FUNCTION "GestMotore" : Void
{ S7_Optimized_Access := 'TRUE' }
VERSION : 0.2
   VAR_INPUT
      K_Motore : Int;
      K_TipoMotore : Int;
      K_Zona : Int;
   END_VAR

   VAR_TEMP
      PI_Mitsubishi : Struct
         STW : Word;
         ActualSpeed : DInt;
         Current : DInt;
         DCBus : DInt;
         AlarmCode : DInt;
         CurrentPeak : DInt;
         DCBusPeak : DInt;
         Appo7 : DInt;
         Appo8 : DInt;
         Appo9 : DInt;
         Appo10 : DInt;
         Appo11 : DInt;
         Appo12 : DInt;
         Appo13 : DInt;
         Appo14 : DInt;
      END_STRUCT;
      PO_Mitsubishi : Struct
         CTW : Word;
         Speed_SP : DInt;
         Acc : DInt;
         Dec : DInt;
         FStart : DInt;
         Appo5 : DInt;
         Appo6 : DInt;
         Appo7 : DInt;
         Appo8 : DInt;
         Appo9 : DInt;
         Appo10 : DInt;
      END_STRUCT;
      PI_Siemens : Struct
         STW : Word;
         ActualSpeed : Int;
         ActualCurrent : Int;
         ActualTorque : Int;
         WarningCode : Int;
         FaultCode : Int;
      END_STRUCT;
      PO_Siemens : Struct
         CTW : Word;
         Speed : Int;
         Spare01 : Int;
         Spare02 : Int;
         Spare03 : Int;
         Spare04 : Int;
      END_STRUCT;
      PI_Schneider : Struct
         STW : Word;
         ActualSpeed : Int;
         Enrgy : Int;
         Segnalaz_Code : Int;
         Spare_01 : Int;
         Spare_02 : Int;
      END_STRUCT;
      PO_Schneider : Struct
         CTW : Word;
         Speed_SP : Int;
         Acc_SP : Int;
         Dec_SP : Int;
         Spare_01 : Int;
         Spare_02 : Int;
      END_STRUCT;
      PI_Movimot : Struct
         STW1 : Word;
         OutputCurrent : Word;
         STW2 : Word;
      END_STRUCT;
      PO_Movimot : Struct
         CTW : Word;
         Speed : Int;
         AccRich : Int;
      END_STRUCT;
      PI_MoviGear : Struct
         STW : Word;
         Actual_Speed : Int;
         Status_Fault : Int;
         Actual_Torque : Int;
         DI : Word;
      END_STRUCT;
      PO_MoviGear : Struct
         CTW : Word;
         Target_Speed : Int;
         Acceleration : Int;
         Deceleration : Int;
         DO : Word;
      END_STRUCT;
      PI_Danfoss : Struct
         STW : Word;
         ActualSpeed : Int;
         CodAllarme_W1 : Int;
         CodAllarme_W2 : Int;
         CodWarning_W1 : Int;
         CodWarning_W2 : Int;
      END_STRUCT;
      PO_Danfoss : Struct
         CTW : Word;
         Speed : Int;
         AccRich : Int;
         DecRich : Int;
         PCD_Spare01 : Int;
         PCD_Spare02 : Int;
      END_STRUCT;
      PI_INVT : Struct
         PKW01 : Word;
         PKW02 : Word;
         PKW03 : Word;
         PKW04 : Word;
         STW : Word;
         ActualSpeed : Int;
         BusVoltage : Int;
         OutputCurrent : Int;
         FaultCode : Int;
         Sapre1 : Int;
         Sapre2 : Int;
         Sapre3 : Int;
      END_STRUCT;
      PO_INVT : Struct
         PKW01 : Word;
         PKW02 : Word;
         PKW03 : Word;
         PKW04 : Word;
         CTW : Word;
         Speed : Int;
         Spare1 : Int;
         Spare2 : Int;
         Spare3 : Int;
         Spare4 : Int;
         Spare5 : Int;
         Spare6 : Int;
      END_STRUCT;
      PI_Movitrac : Struct
         STW1 : Word;
         ActualSpeed : Int;
         ActualCurrent : Word;
      END_STRUCT;
      PO_MoviTrac : Struct
         CTW : Word;
         Speed : Int;
         Reserved : Int;
      END_STRUCT;
      PI_Nidec : Struct
         STW : Word;   // Status Word
         ActualSpeed : DInt;   // Actual Speed
         ActualCurrent : DInt;   // Actual Current
         ActualDCBus : Int;   // Actual Voltage
         FaultCode : USInt;   // Allarm Code
      END_STRUCT;
      PO_Nidec : Struct
         CTW : Word;   // Control Word
         Speed : DInt;   // Speed Request
         RampAcc : DInt;   // Acceleration Ramp Rerquest
         RampDec : DInt;   // Deceleration Ramp Rerquest
      END_STRUCT;
      TempEnc : Struct
         RcvDaEncoderSick : Struct
            ZSW2_ENC : Word;
            G1_ZSW : Word;
            Position01 : DWord;
            Position02 : DWord;
            Speed : DInt;
         END_STRUCT;
         SendAEncoderSick : Struct
            STW2_ENC : Word;
            G1_STW : Word;
         END_STRUCT;
         RcvDaEncoder_Ottico : Struct
            Posizione : DInt;
            Velocita : Int;
         END_STRUCT;
         RcvDaEncoder_Magnetico : Struct
            Posizione : DInt;
         END_STRUCT;
         arrRecord : Array[0..15] of Byte;
         PosizioneLettaEnc : DInt;
         VelocitaLettaEnc : DInt;
         AppoSetupRich : DInt;
         AppoSetupEncoder : UDInt;
         SpazioUltimoCiclo : DInt;
         AppoScrEncoder : DWord;
      END_STRUCT;
      TempTelem : Struct
         RcvDaEncoder : Struct
            M05_IN_ActPos : DWord;
            Status : Struct
               M10Status_IN_AvvPlaus : Bool;
               M10Status_IN_AvvTemp : Bool;
               M10Status_IN_AvvLiv : Bool;
               M10Status_IN_Avvlaser : Bool;
               M10Status_IN_ErrPlaus : Bool;
               M10Status_IN_ErrTemp : Bool;
               M10Status_IN_ErrLiv : Bool;
               M10Status_IN_ErrLaser : Bool;
               M10Status_IN_Spento : Bool;
               M10Status_IN_RiscaldaOn : Bool;
               M10Status_IN_MF1On : Bool;
               M10Status_IN_MF2On : Bool;
               M10Status_IN_Res1 : Bool;
               M10Status_IN_Res2 : Bool;
               M10Status_IN_Res3 : Bool;
               M10Status_IN_NoDist : Bool;
            END_STRUCT;
         END_STRUCT;
         SendAEncode : Struct
            M05_OUT_Preset : DWord;
            Status : Struct
               M10Status_OUT_Res1 : Bool;
               M10Status_OUT_Res2 : Bool;
               M10Status_OUT_Res3 : Bool;
               M10Status_OUT_Res4 : Bool;
               M10Status_OUT_Res5 : Bool;
               M10Status_OUT_Res6 : Bool;
               M10Status_OUT_Res7 : Bool;
               M10Status_OUT_Res8 : Bool;
               M10Status_OUT_Disabil : Bool;
               M10Status_OUT_Res9 : Bool;
               M10Status_OUT_Res10 : Bool;
               M10Status_OUT_Res11 : Bool;
               M10Status_OUT_Res12 : Bool;
               M10Status_OUT_Res13 : Bool;
               M10Status_OUT_Res14 : Bool;
               M10Status_OUT_Res15 : Bool;
            END_STRUCT;
         END_STRUCT;
         arrRecord : Array[0..15] of Byte;
         AppoSetupRich : DInt;
      END_STRUCT;
      ReqDirPos : Bool;
      ReqDirNeg : Bool;
      FunzPositioning : Bool;
      ReqDecBassa : Bool;
      ReqDecStop : Bool;
      ReqStop : Bool;
      ReqCambioVel : Bool;
      CambioPercLavoro : Bool;
      CambioReqVel : Bool;
      CambioReqAcc : Bool;
      CambioReqDec : Bool;
      REQSetup : Bool;
      REQSetupPannello : Bool;
      DistTrgMagPrec : Bool;
      DistTrgMinPrec : Bool;
      RitMotInPrecisione : Bool;
      UnaDirezioneRichiesta : Bool;
      ReqRicTempoProfilo : Bool;
      BloccaAcc : Bool;
      AbilDirPos : Bool;
      AbilDirNeg : Bool;
      SetUpSuSensore : Bool;
      SetUpFermoMeccanico : Bool;
      RichCmdFreno : Bool;
      SpazioFrenoDir : DInt;
      VeloFrenoDir : DInt;
      AppoMoltPrecisione : DInt;
      DecActRich : DInt;
      RicircoloTotale : DInt;
      MezzoRicircoloTotale : DInt;
      DistCambioVel : DInt;
      SpazioStop : DInt;
      SpazioBassa : DInt;
      SpazioCambioVel : DInt;
      DistTRG_ASS : DInt;
      VeloBassaConv : Real;
      SpazioStop_01 : Real;
      SpazioStop_02 : Real;
      SpazioStop_03 : Real;
      SpazioStop_04 : Real;
      SpazioCambioVel_01 : Real;
      SpazioCambioVel_02 : Real;
      VeloProfilo : Real;
      TempoAcc : Real;
      TempoDec_Iniziale : Real;
      TempoDec_Finale : Real;
      TempoVFix : Real;
      K_MotoreInt : Int;
      K_ZonaInt : Int;
      CounterAllarme : Int;
   END_VAR


BEGIN
	REGION Diagnostica programmatore
	    (*Passiamo tutte le costanti di accesso agli array in modo da verificarle e controllarle*)
	    "Diagnostica"(K_Attuale_ArrayInCuiAccediamo := #K_Motore,
	                  K_NumMax_MassimoValoreDellArrayInCuiAccediamo := "K_NumMotore",
	                  K_Tipo_ArrayInCuiAccediamo := "K_TipoMotore",
	                  K_Attuale_DiChiAccede := #K_Motore,
	                  K_Tipo_DiChiAccede := "K_TipoSezionePastorizzatore",
	                  K_AttualeInterno => #K_MotoreInt);

	    "Diagnostica"(K_Attuale_ArrayInCuiAccediamo := #K_Zona,
	                  K_NumMax_MassimoValoreDellArrayInCuiAccediamo := "K_NumZona",
	                  K_Tipo_ArrayInCuiAccediamo := "K_TipoMotore",
	                  K_Attuale_DiChiAccede := #K_Motore,
	                  K_Tipo_DiChiAccede := "K_TipoMotore",
	                  K_AttualeInterno => #K_ZonaInt);
	END_REGION ;
	REGION From inverter
	    CASE "Motore".M[#K_MotoreInt].HW.TipoCollInverter OF
	        1:
	            REGION PN Mitsubishi
	                (*
	                BIT 00: Drive PI:Ready to Switch ON
	                BIT 01: Drive PI:Ready to Operate
	                BIT 02: Drive PI:Operation Enabled
	                BIT 03: Drive PI:Fault Present
	                BIT 04: Drive PI:Coast Stop
	                BIT 05: Drive PI:Quick Stop
	                BIT 06: Drive PI:Switch ON Inhibited
	                BIT 07: Drive PI:Warning
	                BIT 08:
	                BIT 09: Drive PI: Control ON
	                BIT 10:
	                BIT 11:
	                BIT 12:
	                BIT 13:
	                BIT 14:
	                BIT 15:
	                *)
	                "Motore".M[#K_MotoreInt].Dati.RetVal_Read_Inv := DPRD_DAT(LADDR := "Motore".M[#K_MotoreInt].HW.HWIO_Inverter, RECORD => #PI_Mitsubishi);
	                "Motore".M[#K_MotoreInt].In.NoComunInv := ("Motore".M[#K_MotoreInt].Dati.RetVal_Read_Inv OR "Motore".M[#K_MotoreInt].Dati.RetVal_SCR_Inv) <> 0;
	                IF NOT "Motore".M[#K_MotoreInt].In.NoComunInv THEN
	                    (*Appoggio la Status Word per HMI*)
	                    "Motore".M[#K_MotoreInt].HMI.STW1 := #PI_Mitsubishi.STW;
	                    (*Controllo se l'inverter Ã¨ in Fault e relativo Codice*)
	                    "Motore".M[#K_MotoreInt].In.DriverFault := "Zona".Z[#K_Zona].Out.CentralinaOk AND #PI_Mitsubishi.STW.%X3;
	                    IF "Motore".M[#K_MotoreInt].In.DriverFault THEN
	                        "Motore".M[#K_MotoreInt].HMI.CodiceAllarme := #PI_Mitsubishi.AlarmCode;
	                    END_IF;
	                    (* Calcolo La velocitÃ  letta dall'inverter *)
	                    "Motore".M[#K_MotoreInt].Out.MotorSpeed := TRUNC(ABS(DINT_TO_REAL(#PI_Mitsubishi.ActualSpeed)) * DINT_TO_REAL("Motore".M[#K_MotoreInt].Prm.C.VelMax) / 10000.0);
	                    (* Assegno il segnale di Inverter RUN *)
	                    "Motore".M[#K_MotoreInt].In.MotoreRun := #PI_Mitsubishi.STW.%X2;
	                ELSE
	                    (* In caso di mancanza Comunicazione, Azzero i dati *)
	                    "Motore".M[#K_MotoreInt].Out.MotorSpeed := 0;
	                    "Motore".M[#K_MotoreInt].In.MotoreRun := "Motore".M[#K_MotoreInt].In.DriverFault := "Motore".M[#K_MotoreInt].In.DriverWarning := false;
	                END_IF;
	            END_REGION
	        2:
	            REGION PN Siemens
	                (*
	                Definizione Parola di Stato:
	                Bit 00: Drive PI: Ready TO Switch "ON"
	                Bit 01: Drive PI: Ready TO Operate
	                Bit 02: Drive PI: Operation Enabled. The Drive Follows the Setpoint
	                Bit 03: Drive PI: Fault
	                Bit 04: Drive PI: Coast Stop (OFF2) command is NOT Active
	                Bit 05: Drive PI: Quick Stop (OFF3) command is NOT Active
	                Bit 06: Drive PI: Switching on inhibited
	                Bit 07: Drive PI: Warning
	                Bit 08: Drive PI: Setpoint/Actual Value deviation within tolerance range.
	                Bit 09: Drive PI: Master control requested
	                Bit 10: Drive PI: Maximum frequency reached OR exceeded
	                Bit 11: Drive PI: Motor at Current/Torque limit
	                Bit 12: Drive PI: Motor Holding Brake Open
	                Bit 13: Drive PI: Motor Overload
	                Bit 14: Drive PI: Motor Rotation (1 = CW; 0 = CCW).
	                Bit 15: Drive PI: Inverter Overload
	                *)
	                "Motore".M[#K_MotoreInt].Dati.RetVal_Read_Inv := DPRD_DAT(LADDR := "Motore".M[#K_MotoreInt].HW.HWIO_Inverter, RECORD => #PI_Siemens);
	                "Motore".M[#K_MotoreInt].In.NoComunInv := ("Motore".M[#K_MotoreInt].Dati.RetVal_Read_Inv OR "Motore".M[#K_MotoreInt].Dati.RetVal_SCR_Inv) <> 0;
	                IF NOT "Motore".M[#K_MotoreInt].In.NoComunInv THEN
	                    (*Appoggio la Status Word per HMI*)
	                    "Motore".M[#K_MotoreInt].HMI.STW1 := #PI_Siemens.STW;
	                    (*Controllo se l'inverter Ã¨ in Fault e relativo Codice*)
	                    "Motore".M[#K_MotoreInt].In.DriverFault := "Zona".Z[#K_Zona].Out.CentralinaOk AND (#PI_Siemens.STW.%X3 OR NOT #PI_Siemens.STW.%X9);
	                    IF "Motore".M[#K_MotoreInt].In.DriverFault THEN
	                        "Motore".M[#K_MotoreInt].HMI.CodiceAllarme := #PI_Siemens.FaultCode;
	                    END_IF;
	                    (*Controllo se l'inverter Ã¨ in Warning e relativo Codice*)
	                    "Motore".M[#K_MotoreInt].In.DriverWarning := "Zona".Z[#K_Zona].Out.CentralinaOk AND #PI_Siemens.STW.%X7;
	                    IF "Motore".M[#K_MotoreInt].In.DriverWarning THEN
	                        "Motore".M[#K_MotoreInt].HMI.CodiceWarning := #PI_Siemens.WarningCode;
	                    END_IF;
	                    (* Calcolo La velocitÃ  letta dall'inverter *)
	                    "Motore".M[#K_MotoreInt].Out.MotorSpeed := INT_TO_DINT(#PI_Siemens.ActualSpeed) * "Motore".M[#K_MotoreInt].Prm.C.VelMax / 16384;
	                    (* Assegno il segnale di Inverter RUN *)
	                    "Motore".M[#K_MotoreInt].In.MotoreRun := #PI_Siemens.STW.%X2;
	                ELSE
	                    (* In caso di mancanza Comunicazione, Azzero i dati *)
	                    "Motore".M[#K_MotoreInt].Out.MotorSpeed := 0;
	                    "Motore".M[#K_MotoreInt].In.MotoreRun := "Motore".M[#K_MotoreInt].In.DriverFault := "Motore".M[#K_MotoreInt].In.DriverWarning := false;
	                END_IF;
	            END_REGION
	        3:
	            REGION PN_Schneider
	                (*
	                BIT 00: Drive PI: Mains power supply is switched on, electronics are initialized, pulses are inhibited
	                BIT 01: Drive PI: Refer to control word 1, bit 0
	                BIT 02: Drive PI: Drive follows a reference frequency.
	                BIT 03: Drive PI: An error has been detected.
	                BIT 04: Drive PI: 1= --, 0= Coast stop (OFF 2) command is present
	                BIT 05: Drive PI: 1= --, 0= Quick Stop (OFF 3) command is present.
	                BIT 06: Drive PI: The drive is in Switching on inhibited operating state.
	                BIT 07: Drive PI: Warning information present in the service/maintenance parameter, acknowledgement required.
	                BIT 08: Actual value is within a tolerance band; dynamic speed discrepancies are permissible.
	                BIT 09: The automation system controls the drive.
	                BIT 10: Actual output frequency â‰¥ reference frequency which may be set via the parameter number.
	                BIT 11: Drive PI: Reserved
	                BIT 12: Drive PI: Reserved
	                BIT 13: Drive PI: Reserved
	                BIT 14: Drive PI: Reserved
	                BIT 15: Drive PI: Reserved
	                *)
	                "Motore".M[#K_MotoreInt].Dati.RetVal_Read_Inv := DPRD_DAT(LADDR := "Motore".M[#K_MotoreInt].HW.HWIO_Inverter, RECORD => #PI_Schneider);
	                "Motore".M[#K_MotoreInt].In.NoComunInv := ("Motore".M[#K_MotoreInt].Dati.RetVal_Read_Inv OR "Motore".M[#K_MotoreInt].Dati.RetVal_SCR_Inv) <> 0;
	                IF NOT "Motore".M[#K_MotoreInt].In.NoComunInv THEN
	                    (*Appoggio la Status Word per HMI*)
	                    "Motore".M[#K_MotoreInt].HMI.STW1 := #PI_Schneider.STW;
	                    (*Controllo se l'inverter Ã¨ in Fault e relativo Codice*)
	                    "Motore".M[#K_MotoreInt].In.DriverFault := "Zona".Z[#K_Zona].Out.CentralinaOk AND #PI_Schneider.STW.%X3;
	                    IF "Motore".M[#K_MotoreInt].In.DriverFault THEN
	                        "Motore".M[#K_MotoreInt].HMI.CodiceAllarme := #PI_Schneider.Segnalaz_Code;
	                    END_IF;
	                    // Inverter in warning
	                    "Motore".M[#K_MotoreInt].In.DriverWarning := "Zona".Z[#K_Zona].Out.CentralinaOk AND #PI_Schneider.STW.%X7;
	                    IF "Motore".M[#K_MotoreInt].In.DriverWarning THEN
	                        "Motore".M[#K_MotoreInt].HMI.CodiceWarning := #PI_Schneider.Spare_01;
	                    END_IF;
	                    (* Calcolo La velocitÃ  letta dall'inverter *)
	                    "Motore".M[#K_MotoreInt].Out.MotorSpeed := ABS(INT_TO_DINT(#PI_Schneider.ActualSpeed) * "Motore".M[#K_MotoreInt].Prm.C.VelMax / 3000);
	                    (* Assegno il segnale di Inverter RUN *)
	                    "Motore".M[#K_MotoreInt].In.MotoreRun := #PI_Schneider.STW.%X2;
	                ELSE
	                    (* In caso di mancanza Comunicazione, Azzero i dati *)
	                    "Motore".M[#K_MotoreInt].Out.MotorSpeed := 0;
	                    "Motore".M[#K_MotoreInt].In.MotoreRun := "Motore".M[#K_MotoreInt].In.DriverFault := "Motore".M[#K_MotoreInt].In.DriverWarning := false;
	                END_IF;
	            END_REGION
	        4:
	            REGION PN Movimot
	                (*
	                Status Word 01

	                BIT 08: Alarm Code Bit 00
	                BIT 09: Alarm Code Bit 01
	                BIT 10: Alarm Code Bit 02
	                BIT 11: Alarm Code Bit 03
	                BIT 12: Alarm Code Bit 04
	                BIT 13: Alarm Code Bit 05
	                BIT 14: Alarm Code Bit 06
	                BIT 15: Alarm Code Bit 07
	                BIT 00: 0=Control Not Enabled / 1=Enabled
	                BIT 01: 0=Inverter Not Ready / 1=Ready
	                BIT 02: 0=PO Data Not Enabled / 1=Enabled
	                BIT 03: Reserved
	                BIT 04: Reserved
	                BIT 05: 0=OK / 1=Malfunction/Warning
	                BIT 06: Reserved
	                BIT 07: Reserved

	                Status Word 02

	                BIT 08: 0=Brake Released / 1= Brake Applied
	                BIT 09: 0=Not Ready For Operation / 1=Ready
	                BIT 10: 0=Stop / 1=Motor Run CW
	                BIT 11: 0=Stop / 1=Motor Run CCW
	                BIT 12: 0=Stop / 1=Set Point F2
	                BIT 13: Reserved
	                BIT 14: Reserved
	                BIT 15: Reserved
	                BIT 00: 0=Control Not Enabled / 1=Enabled
	                BIT 01: 0=Inverter Not Ready / 1=Ready
	                BIT 02: 0=PO Data Not Enabled / 1=Enabled
	                BIT 03: Reserved
	                BIT 04: Reserved
	                BIT 05: 0=OK / 1=Malfunction/Warning
	                BIT 06: Reserved
	                BIT 07: Reserved
	                *)
	                "Motore".M[#K_MotoreInt].Dati.RetVal_Read_Inv := DPRD_DAT(LADDR := "Motore".M[#K_MotoreInt].HW.HWIO_Inverter, RECORD => #PI_Movimot);
	                "Motore".M[#K_MotoreInt].In.NoComunInv := ("Motore".M[#K_MotoreInt].Dati.RetVal_Read_Inv OR "Motore".M[#K_MotoreInt].Dati.RetVal_SCR_Inv) <> 0;
	                IF NOT "Motore".M[#K_MotoreInt].In.NoComunInv THEN
	                    (*Appoggio la Status Word per HMI*)
	                    "Motore".M[#K_MotoreInt].HMI.STW1 := #PI_Movimot.STW1;
	                    "Motore".M[#K_MotoreInt].HMI.STW2 := #PI_Movimot.OutputCurrent;
	                    "Motore".M[#K_MotoreInt].HMI.STW3 := #PI_Movimot.STW2;
	                    (* Controllo Stato Sezionatore Aperto *)
	                    "Motore".M[#K_MotoreInt].In.SezAperto := FALSE;
	                    IF #PI_Movimot.STW1.%X5 AND #PI_Movimot.STW1.%X8 AND #PI_Movimot.STW1.%X9 AND #PI_Movimot.STW1.%X10 AND
	                        #PI_Movimot.STW1.%X11 AND NOT #PI_Movimot.STW1.%X12 AND #PI_Movimot.STW1.%X13 AND #PI_Movimot.STW1.%X14 AND
	                        NOT #PI_Movimot.STW1.%X15 AND "Zona".Z[#K_Zona].Out.CentralinaOk THEN
	                        IF "Motore".M[#K_MotoreInt].Dati.ContOffSezAperto < 0 THEN
	                            "Motore".M[#K_MotoreInt].In.SezAperto := TRUE;
	                        ELSE
	                            "Motore".M[#K_MotoreInt].Dati.ContOffSezAperto -= REAL_TO_INT("Zona".Comuni.TempoCicloCpu_r);
	                        END_IF;
	                    ELSE
	                        "Motore".M[#K_MotoreInt].Dati.ContOffSezAperto := 4000;
	                    END_IF;
	                    (*Controllo se l'inverter Ã¨ in Fault e relativo Codice*)
	                    "Motore".M[#K_MotoreInt].In.DriverFault := "Zona".Z[#K_Zona].Out.CentralinaOk AND NOT "Motore".M[#K_MotoreInt].In.SezAperto AND (#PI_Movimot.STW1.%X5 OR NOT #PI_Movimot.STW1.%X1 OR NOT #PI_Movimot.STW1.%X2);
	                    IF "Motore".M[#K_MotoreInt].In.DriverFault THEN
	                        "Motore".M[#K_MotoreInt].HMI.CodiceAllarme := #PI_Movimot.STW1.%B1;
	                    END_IF;
	                    (* Calcolo La velocitÃ  letta dall'inverter *)
	                    "Motore".M[#K_MotoreInt].Out.MotorSpeed := TRUNC("Motore".M[#K_MotoreInt].Out.Vel);
	                    (* Assegno il segnale di Inverter RUN *)
	                    "Motore".M[#K_MotoreInt].In.MotoreRun := #PI_Movimot.STW1.%X0 AND #PI_Movimot.STW2.%X1;
	                ELSE
	                    (* In caso di mancanza Comunicazione, Azzero i dati *)
	                    "Motore".M[#K_MotoreInt].Out.MotorSpeed := 0;
	                    "Motore".M[#K_MotoreInt].In.MotoreRun := "Motore".M[#K_MotoreInt].In.DriverFault := "Motore".M[#K_MotoreInt].In.DriverWarning := false;
	                END_IF;
	            END_REGION
	        5:
	            REGION PN MoviGear
	                (*
	                BIT 00: Ready
	                BIT 01: STO Disattivato
	                BIT 02: Output Stage Pronto
	                BIT 03: Freno Rilasciato
	                BIT 04: Motore in movimento
	                BIT 05: Motore Riferenziato
	                BIT 06: Nuova posizione Relativa Applicata
	                BIT 07: In Posizione
	                BIT 08: Fault
	                BIT 09: Warning
	                BIT 10: Attivato Motore 2
	                BIT 11: VelocitÃ  Attuale = A Target
	                BIT 12: Limiti SW Disattivati
	                BIT 13: Riservato
	                BIT 14: Stand By Attivo
	                BIT 15: HandShake
	                *)
	                "Motore".M[#K_MotoreInt].Dati.RetVal_Read_Inv := DPRD_DAT(LADDR := "Motore".M[#K_MotoreInt].HW.HWIO_Inverter, RECORD => #PI_MoviGear);
	                "Motore".M[#K_MotoreInt].In.NoComunInv := ("Motore".M[#K_MotoreInt].Dati.RetVal_Read_Inv OR "Motore".M[#K_MotoreInt].Dati.RetVal_SCR_Inv) <> 0;
	                IF NOT "Motore".M[#K_MotoreInt].In.NoComunInv THEN
	                    (*Appoggio la Status Word per HMI*)
	                    "Motore".M[#K_MotoreInt].HMI.STW1 := #PI_MoviGear.STW;
	                    (*Controllo se l'inverter Ã¨ in Fault e relativo Codice*)
	                    "Motore".M[#K_MotoreInt].In.DriverFault := "Zona".Z[#K_Zona].Out.CentralinaOk AND (#PI_MoviGear.STW.%X8 OR NOT #PI_MoviGear.STW.%X0);
	                    IF "Motore".M[#K_MotoreInt].In.DriverFault THEN
	                        IF NOT #PI_MoviGear.STW.%X0 THEN
	                            "Motore".M[#K_MotoreInt].HMI.CodiceAllarme := #PI_MoviGear.Status_Fault;
	                        ELSE
	                            "Motore".M[#K_MotoreInt].HMI.CodiceAllarme := 1;
	                        END_IF;
	                    END_IF;
	                    (*Controllo se l'inverter Ã¨ in Warning e relativo Codice*)
	                    "Motore".M[#K_MotoreInt].In.DriverWarning := "Zona".Z[#K_Zona].Out.CentralinaOk AND #PI_MoviGear.STW.%X9;
	                    IF "Motore".M[#K_MotoreInt].In.DriverWarning THEN
	                        "Motore".M[#K_MotoreInt].HMI.CodiceWarning := "Motore".M[#K_MotoreInt].HMI.CodiceWarning;
	                    END_IF;
	                    (* Calcolo La velocitÃ  letta dall'inverter *)
	                    "Motore".M[#K_MotoreInt].Out.MotorSpeed := ABS(INT_TO_DINT(#PI_MoviGear.Actual_Speed)) * "Motore".M[#K_MotoreInt].Prm.C.VelMax / 3000;
	                    (* Assegno il segnale di Inverter RUN *)
	                    "Motore".M[#K_MotoreInt].In.MotoreRun := #PI_MoviGear.STW.%X0 AND #PI_MoviGear.STW.%X2;
	                ELSE
	                    (* In caso di mancanza Comunicazione, Azzero i dati *)
	                    "Motore".M[#K_MotoreInt].Out.MotorSpeed := 0;
	                    "Motore".M[#K_MotoreInt].In.MotoreRun := "Motore".M[#K_MotoreInt].In.DriverFault := "Motore".M[#K_MotoreInt].In.DriverWarning := false;
	                END_IF;
	            END_REGION
	        6:
	            REGION PN Danfoss
	                (*
	                BIT 00: 0=Control NOT Ready       1=Ready
	                BIT 01: 0=Drive NOT Ready       1=Ready
	                BIT 02: 0=Coasting        1=Enable
	                BIT 03: 0=No error        1=Trip
	                BIT 04: OFF/ON 2
	                BIT 05: OFF/ON 3
	                BIT 06: 0=Start possible        1=NOT possible
	                BIT 07: 0=No warning        1=Warning
	                BIT 08: 0= Speed><REF       1= Speed=REF
	                BIT 09: 0=Local oper       1=Bus control
	                BIT 10: 0=Out Freq.Limit     1=Freq.Limit OK
	                BIT 11: 0=No operation      1=In operation
	                BIT 12: 0=Drive OK       1=Stopped, Autostart
	                BIT 13: 0=Voltage OK       1=Voltage exceeded
	                BIT 14: 0=OFF      1=Comparatore 0 ON
	                BIT 15: 0=OFF      1=Comparatore 1 ON
	                *)
	                "Motore".M[#K_MotoreInt].Dati.RetVal_Read_Inv := DPRD_DAT(LADDR := "Motore".M[#K_MotoreInt].HW.HWIO_Inverter, RECORD => #PI_Danfoss);
	                "Motore".M[#K_MotoreInt].In.NoComunInv := ("Motore".M[#K_MotoreInt].Dati.RetVal_Read_Inv OR "Motore".M[#K_MotoreInt].Dati.RetVal_SCR_Inv) <> 0;
	                IF NOT "Motore".M[#K_MotoreInt].In.NoComunInv THEN
	                    (*Appoggio la Status Word per HMI*)
	                    "Motore".M[#K_MotoreInt].HMI.STW1 := #PI_Danfoss.STW;
	                    (*Controllo se l'inverter Ã¨ in Fault e relativo Codice*)
	                    "Motore".M[#K_MotoreInt].In.DriverFault := "Zona".Z[#K_Zona].Out.CentralinaOk AND (#PI_Danfoss.STW.%X3 OR NOT #PI_Danfoss.STW.%X9);
	                    IF "Motore".M[#K_MotoreInt].In.DriverFault THEN
	                        "Motore".M[#K_MotoreInt].HMI.CodiceAllarme := #PI_Danfoss.CodAllarme_W2 OR SHL(IN := #PI_Danfoss.CodAllarme_W1, N := 16);
	                    END_IF;
	                    (*Controllo se l'inverter Ã¨ in Warning e relativo Codice*)
	                    "Motore".M[#K_MotoreInt].In.DriverWarning := "Zona".Z[#K_Zona].Out.CentralinaOk AND #PI_Danfoss.STW.%X7;
	                    IF "Motore".M[#K_MotoreInt].In.DriverWarning THEN
	                        "Motore".M[#K_MotoreInt].HMI.CodiceAllarme := #PI_Danfoss.CodWarning_W2 OR SHL(IN := #PI_Danfoss.CodWarning_W1, N := 16);
	                    END_IF;
	                    (* Calcolo La velocitÃ  letta dall'inverter *)
	                    "Motore".M[#K_MotoreInt].Out.MotorSpeed := ABS(INT_TO_DINT(#PI_Danfoss.ActualSpeed)) * "Motore".M[#K_MotoreInt].Prm.C.VelMax / 16384;
	                    (* Assegno il segnale di Inverter RUN *)
	                    "Motore".M[#K_MotoreInt].In.MotoreRun := #PI_Danfoss.STW.%X2 AND #PI_Danfoss.STW.%X11;
	                ELSE
	                    (* In caso di mancanza Comunicazione, Azzero i dati *)
	                    "Motore".M[#K_MotoreInt].Out.MotorSpeed := 0;
	                    "Motore".M[#K_MotoreInt].In.MotoreRun := "Motore".M[#K_MotoreInt].In.DriverFault := "Motore".M[#K_MotoreInt].In.DriverWarning := false;
	                END_IF;
	            END_REGION
	        7:
	            REGION PN Movitrac
	                (*
	                Status Word 01

	                BIT 08: Alarm Code Bit 00
	                BIT 09: Alarm Code Bit 01
	                BIT 10: Alarm Code Bit 02
	                BIT 11: Alarm Code Bit 03
	                BIT 12: Alarm Code Bit 04
	                BIT 13: Alarm Code Bit 05
	                BIT 14: Alarm Code Bit 06
	                BIT 15: Alarm Code Bit 07
	                BIT 00: 0=Control Not Enabled / 1=Enabled
	                BIT 01: 0=Inverter Not Ready / 1=Ready
	                BIT 02: 0=PO Data Not Enabled / 1=Enabled
	                BIT 03: Reserved
	                BIT 04: Reserved
	                BIT 05: 0=OK / 1=Malfunction/Warning
	                BIT 06: Reserved
	                BIT 07: Reserved
	                *)
	                "Motore".M[#K_MotoreInt].Dati.RetVal_Read_Inv := DPRD_DAT(LADDR := "Motore".M[#K_MotoreInt].HW.HWIO_Inverter, RECORD => #PI_Movitrac);
	                "Motore".M[#K_MotoreInt].In.NoComunInv := ("Motore".M[#K_MotoreInt].Dati.RetVal_Read_Inv OR "Motore".M[#K_MotoreInt].Dati.RetVal_SCR_Inv) <> 0;
	                IF NOT "Motore".M[#K_MotoreInt].In.NoComunInv THEN
	                    (*Appoggio la Status Word per HMI*)
	                    "Motore".M[#K_MotoreInt].HMI.STW1 := #PI_Movitrac.STW1;
	                    (*Controllo se l'inverter Ã¨ in Fault e relativo Codice*)
	                    "Motore".M[#K_MotoreInt].In.DriverFault := "Zona".Z[#K_Zona].Out.CentralinaOk AND (#PI_Movitrac.STW1.%X5 OR NOT #PI_Movitrac.STW1.%X1 OR NOT #PI_Movitrac.STW1.%X2);
	                    IF "Motore".M[#K_MotoreInt].In.DriverFault THEN
	                        "Motore".M[#K_MotoreInt].HMI.CodiceAllarme := #PI_Movitrac.STW1.%B1;
	                    END_IF;
	                    (* Calcolo La velocitÃ  letta dall'inverter *)
	                    "Motore".M[#K_MotoreInt].Out.MotorSpeed := ABS(INT_TO_DINT(#PI_Movitrac.ActualSpeed)) * "Motore".M[#K_MotoreInt].Prm.C.VelMax / 16384;
	                    (* Assegno il segnale di Inverter RUN *)
	                    "Motore".M[#K_MotoreInt].In.MotoreRun := #PI_Movitrac.STW1.%X0;
	                ELSE
	                    (* In caso di mancanza Comunicazione, Azzero i dati *)
	                    "Motore".M[#K_MotoreInt].Out.MotorSpeed := 0;
	                    "Motore".M[#K_MotoreInt].In.MotoreRun := "Motore".M[#K_MotoreInt].In.DriverFault := "Motore".M[#K_MotoreInt].In.DriverWarning := false;
	                END_IF;
	            END_REGION
	        8:
	            REGION PN INVT
	                (*
	                Bit   Descr
	                0â€“7     Running state
	                Value   Desc
	                1       Forward running
	                2       Reverse running
	                3       Stopped
	                4       Faulty
	                5       POFF
	                Bit:8 Bus voltage established: 0=Not ready to Run, 1=Ready to Run
	                Bit 9â€“10: Motor group feedback
	                BIT 11: 0=Asynchronous Motor 1=Syncronous Motor
	                BIT 12:Overload pre-alarm feedback  0=No overload pre-alarm generated 1=Overload pre-alarm generated
	                Bit     Descr
	                13â€“14   Run/Stop mode
	                Value   Desc
	                0       Keypad-based control
	                1       Terminal-based control
	                2       Communication-based control
	                3       Reserved
	                BIT 15Heartbeat feedback : 0=OFF      1=Comparatore 1 ON
	                *)
	                "Motore".M[#K_MotoreInt].Dati.RetVal_Read_Inv := DPRD_DAT(LADDR := "Motore".M[#K_MotoreInt].HW.HWIO_Inverter, RECORD => #PI_INVT);
	                "Motore".M[#K_MotoreInt].In.NoComunInv := ("Motore".M[#K_MotoreInt].Dati.RetVal_Read_Inv OR "Motore".M[#K_MotoreInt].Dati.RetVal_SCR_Inv) <> 0;
	                IF NOT "Motore".M[#K_MotoreInt].In.NoComunInv THEN
	                    (*Appoggio la Status Word per HMI*)
	                    "Motore".M[#K_MotoreInt].HMI.STW1 := #PI_INVT.STW;
	                    (*Controllo se l'inverter Ã¨ in Fault e relativo Codice*)
	                    "Motore".M[#K_MotoreInt].In.DriverFault := #PI_INVT.STW.%B0 = 4 AND "Zona".Z[#K_Zona].Out.CentralinaOk;
	                    IF "Motore".M[#K_MotoreInt].In.DriverFault THEN
	                        "Motore".M[#K_MotoreInt].HMI.CodiceAllarme := #PI_INVT.FaultCode;
	                    END_IF;
	                    (*Controllo se l'inverter Ã¨ in Warning e relativo Codice*)
	                    "Motore".M[#K_MotoreInt].In.DriverWarning := #PI_INVT.STW.%X12;
	                    (* Calcolo La velocitÃ  letta dall'inverter *)
	                    "Motore".M[#K_MotoreInt].Out.MotorSpeed := ABS(INT_TO_DINT(#PI_INVT.ActualSpeed)) * "Motore".M[#K_MotoreInt].Prm.C.VelMax / 10000;
	                    (* Assegno il segnale di Inverter RUN *)
	                    "Motore".M[#K_MotoreInt].In.MotoreRun := #PI_INVT.STW.%X8;
	                ELSE
	                    (* In caso di mancanza Comunicazione, Azzero i dati *)
	                    "Motore".M[#K_MotoreInt].Out.MotorSpeed := 0;
	                    "Motore".M[#K_MotoreInt].In.MotoreRun := "Motore".M[#K_MotoreInt].In.DriverFault := "Motore".M[#K_MotoreInt].In.DriverWarning := false;
	                END_IF;
	            END_REGION
	        9:
	            REGION NIDEC
	                (*
	                BIT 00: Drive Healthy
	                BIT 01: Drive Active
	                BIT 02: Zero Frequency
	                BIT 03: Running At OR Below Minimum Frequency
	                BIT 04: Below Set Frequency
	                BIT 05: At Frequency
	                BIT 06: Above Set Frequency
	                BIT 07: Rated Load Reached
	                BIT 08: Current Limit Active
	                BIT 09: Regenerating
	                BIT 10: Braking IGBT Active
	                BIT 11: Braking Resistor Alarm
	                BIT 12: Reverse Direction Commanded
	                BIT 13: Reverse Direction Running
	                BIT 14: Supply Loss
	                *)
	                IF NOT "Motore".M[#K_MotoreInt].In.NoComunInv THEN
	                    //VariantGet(SRC := #PI_Inv, DST => #PI_Nidec);
	                    "Motore".M[#K_MotoreInt].HMI.STW1 := #PI_Nidec.STW;
	                    (*Controllo se l'inverter Ã¨ in Fault e relativo Codice*)
	                    "Motore".M[#K_MotoreInt].In.DriverFault := NOT #PI_Nidec.STW.%X0 AND "Zona".Z[#K_Zona].Out.CentralinaOk;
	                    IF "Motore".M[#K_MotoreInt].In.DriverFault THEN
	                        "Motore".M[#K_MotoreInt].HMI.CodiceAllarme := #PI_Nidec.FaultCode;
	                    END_IF;
	                    (* Calcolo La velocitÃ  letta dall'inverter *)
	                    "Motore".M[#K_MotoreInt].Out.MotorSpeed := ABS(#PI_Nidec.ActualSpeed) * "Motore".M[#K_MotoreInt].Prm.C.VelMax / 10000;
	                    (* Assegno il segnale di Inverter RUN *)
	                    "Motore".M[#K_MotoreInt].In.MotoreRun := #PI_Nidec.STW.%X1;
	                ELSE
	                    "Motore".M[#K_MotoreInt].Out.MotorSpeed := 0;
	                    "Motore".M[#K_MotoreInt].In.MotoreRun := "Motore".M[#K_MotoreInt].In.DriverFault := "Motore".M[#K_MotoreInt].In.DriverWarning := false;
	                END_IF;
	            END_REGION
	    END_CASE;
	END_REGION
	REGION Encoder manager
	    IF "Zona".Z[#K_Zona].Out.Auto THEN
	        "Motore".M[#K_MotoreInt].HMI.Setup := "Motore".M[#K_MotoreInt].HMI.ManMov := false;
	        "Motore".M[#K_MotoreInt].HMI.ModoInizializza := 0;
	    END_IF;
	    REGION Calcolo Target Position Teorica
	        #RicircoloTotale := "Motore".M[#K_MotoreInt].Prm.Enc.ModuloPosEnc - "Motore".M[#K_MotoreInt].Prm.Enc.ModuloNegEnc;
	        #MezzoRicircoloTotale := #RicircoloTotale / 2;
	        IF "Motore".M[#K_MotoreInt].Out.InMarcia THEN
	            "Motore".M[#K_MotoreInt].Prm.C.TrgPos += "Motore".M[#K_MotoreInt].Out.Vel * "Zona".Comuni.TempoCicloCpu_r / 1000.0;
	            "Motore".M[#K_MotoreInt].Dati.TrgPosDint := TRUNC("Motore".M[#K_MotoreInt].Prm.C.TrgPos);
	            IF "Motore".M[#K_MotoreInt].Prm.Mech.EndLess THEN
	                IF "Motore".M[#K_MotoreInt].Dati.TrgPosDint < "Motore".M[#K_MotoreInt].Prm.Enc.ModuloNegEnc THEN
	                    // Aggiorno l'ultima posizione di target memorizzata
	                    "Motore".M[#K_MotoreInt].Prm.C.TrgPos += DINT_TO_REAL(#RicircoloTotale);
	                    "Motore".M[#K_MotoreInt].Dati.TrgPosDint := "Motore".M[#K_MotoreInt].Dati.OldTrgPosDint := TRUNC("Motore".M[#K_MotoreInt].Prm.C.TrgPos);
	                ELSIF "Motore".M[#K_MotoreInt].Dati.TrgPosDint > "Motore".M[#K_MotoreInt].Prm.Enc.ModuloPosEnc THEN
	                    "Motore".M[#K_MotoreInt].Prm.C.TrgPos -= DINT_TO_REAL(#RicircoloTotale);
	                    "Motore".M[#K_MotoreInt].Dati.TrgPosDint := "Motore".M[#K_MotoreInt].Dati.OldTrgPosDint := TRUNC("Motore".M[#K_MotoreInt].Prm.C.TrgPos);
	                END_IF;
	            END_IF;
	            IF "Motore".M[#K_MotoreInt].Prm.Enc.EncoderLess THEN
	                "Motore".M[#K_MotoreInt].Out.ActPos := "Motore".M[#K_MotoreInt].Dati.TrgPosDint;
	                "Motore".M[#K_MotoreInt].Prm.C.EncPos := "Motore".M[#K_MotoreInt].Prm.C.TrgPos;
	            END_IF;
	        END_IF;
	    END_REGION
	    REGION Condizioni Setup Encoder
	        IF "Motore".M[#K_MotoreInt].In.Setup THEN
	            #REQSetup := TRUE;
	        ELSIF "Motore".M[#K_MotoreInt].HMI.Setup THEN
	            #REQSetupPannello := "Motore".M[#K_MotoreInt].HMI.PulsanteSetupPremuto AND "Zona".Z[#K_Zona].Gen.Reset;
	            IF #REQSetupPannello THEN
	                "Motore".M[#K_MotoreInt].Out.EncoderHomed := FALSE;
	                #SetUpSuSensore := "Motore".M[#K_MotoreInt].Prm.Enc.SetupMode = 2 OR "Motore".M[#K_MotoreInt].Prm.Enc.SetupMode = 10;
	                #SetUpFermoMeccanico := "Motore".M[#K_MotoreInt].Prm.Enc.SetupMode = 4 OR "Motore".M[#K_MotoreInt].Prm.Enc.SetupMode = 12;
	                IF NOT #SetUpSuSensore AND NOT #SetUpFermoMeccanico THEN
	                    #REQSetup := TRUE;
	                    "Motore".M[#K_MotoreInt].Allarmi.SetupEncoderEseg := TRUE;
	                END_IF;
	            END_IF;
	        END_IF;
	    END_REGION
	    REGION Setup Su Sensore
	        IF #SetUpSuSensore OR "Motore".M[#K_MotoreInt].Dati.SetupSensoreTrovato THEN
	            REGION Tempo OFF Marcia Motore
	                IF NOT "Motore".M[#K_MotoreInt].Dati.MotoreFermo THEN
	                    "Motore".M[#K_MotoreInt].Dati.ContTOffMotoreMarcia := 1000;
	                    "Motore".M[#K_MotoreInt].Dati.TOffMotoreMarcia := true;
	                ELSE
	                    IF "Motore".M[#K_MotoreInt].Dati.ContTOffMotoreMarcia > 0 THEN
	                        "Motore".M[#K_MotoreInt].Dati.ContTOffMotoreMarcia -= REAL_TO_INT("Zona".Comuni.TempoCicloCpu_r);
	                    ELSE
	                        "Motore".M[#K_MotoreInt].Dati.TOffMotoreMarcia := false;
	                    END_IF;
	                END_IF;
	            END_REGION ;
	            #REQSetup := "Motore".M[#K_MotoreInt].Out.SetUpSensEseg := "Motore".M[#K_MotoreInt].Dati.SetupSensoreTrovato AND NOT "Motore".M[#K_MotoreInt].Dati.TOffMotoreMarcia;
	            IF #REQSetup THEN
	                "Motore".M[#K_MotoreInt].Allarmi.SetupEncoderEseg := TRUE;
	            END_IF;
	            IF "Motore".M[#K_MotoreInt].Out.SetUpSensEseg THEN
	                IF NOT "Motore".M[#K_MotoreInt].Dati.AppoImpEsecSetUP THEN
	                    "Motore".M[#K_MotoreInt].Dati.Encoder.ValoKSetupSuSens := "Motore".M[#K_MotoreInt].Out.ActPos - "Motore".M[#K_MotoreInt].Dati.PosImpulsoSetup;
	                    "Motore".M[#K_MotoreInt].Dati.AppoImpEsecSetUP := TRUE;
	                END_IF;
	            ELSE
	                "Motore".M[#K_MotoreInt].Dati.AppoImpEsecSetUP := FALSE;
	            END_IF;
	            IF "Motore".M[#K_MotoreInt].Out.SetUpSensEseg AND NOT #SetUpSuSensore THEN
	                IF "Motore".M[#K_MotoreInt].Dati.ContSetUPEncoder > 300 THEN
	                    "Motore".M[#K_MotoreInt].Dati.SetupSensoreTrovato := false;
	                ELSE
	                    "Motore".M[#K_MotoreInt].Dati.ContSetUPEncoder += REAL_TO_INT("Zona".Comuni.TempoCicloCpu_r);
	                END_IF;
	            ELSE
	                "Motore".M[#K_MotoreInt].Dati.ContSetUPEncoder := 0;
	            END_IF;
	            IF NOT "Motore".M[#K_MotoreInt].Dati.SetupSensoreTrovato THEN
	                IF NOT "Motore".M[#K_MotoreInt].In.SensAzz THEN
	                    IF ("Motore".M[#K_MotoreInt].Prm.Enc.SetupMode = 2 AND "Motore".M[#K_MotoreInt].Dati.ActVelNeg) OR
	                        ("Motore".M[#K_MotoreInt].Prm.Enc.SetupMode = 10 AND "Motore".M[#K_MotoreInt].Dati.ActVelPos) THEN
	                        "Motore".M[#K_MotoreInt].Dati.SetupSensoreTrovato := true;
	                        "Motore".M[#K_MotoreInt].Dati.PosImpulsoSetup := "Motore".M[#K_MotoreInt].Out.ActPos;
	                    END_IF;
	                ELSIF ("Motore".M[#K_MotoreInt].Prm.Enc.SetupMode = 2 AND "Motore".M[#K_MotoreInt].Out.ActDirPos) OR
	                    ("Motore".M[#K_MotoreInt].Prm.Enc.SetupMode = 10 AND "Motore".M[#K_MotoreInt].Out.ActDirNeg) THEN
	                    "Motore".M[#K_MotoreInt].Dati.ContTimeOutAzzeramento := 0;
	                END_IF;
	                "Motore".M[#K_MotoreInt].In.CmdPosRich := ("Motore".M[#K_MotoreInt].Prm.Enc.SetupMode = 2 AND NOT "Motore".M[#K_MotoreInt].In.SensAzz) OR ("Motore".M[#K_MotoreInt].Prm.Enc.SetupMode = 10 AND "Motore".M[#K_MotoreInt].In.SensAzz);
	                "Motore".M[#K_MotoreInt].In.CmdNegRich := ("Motore".M[#K_MotoreInt].Prm.Enc.SetupMode = 10 AND NOT "Motore".M[#K_MotoreInt].In.SensAzz) OR ("Motore".M[#K_MotoreInt].Prm.Enc.SetupMode = 2 AND "Motore".M[#K_MotoreInt].In.SensAzz);
	                IF "Motore".M[#K_MotoreInt].In.CmdPosRich THEN
	                    "Motore".M[#K_MotoreInt].In.CmdVelocitaRich := "Motore".M[#K_MotoreInt].Prm.VelSgancioFrenoPos;
	                ELSIF "Motore".M[#K_MotoreInt].In.CmdNegRich THEN
	                    "Motore".M[#K_MotoreInt].In.CmdVelocitaRich := "Motore".M[#K_MotoreInt].Prm.VelSgancioFrenoNeg;
	                END_IF;
	            ELSE
	                "Motore".M[#K_MotoreInt].In.CmdPosRich := "Motore".M[#K_MotoreInt].In.CmdNegRich := "Motore".M[#K_MotoreInt].In.Positioning := false;
	            END_IF;
	        END_IF;
	    END_REGION
	    REGION SetupSuFermoMeccanico
	        IF #SetUpFermoMeccanico OR "Motore".M[#K_MotoreInt].Dati.SetupFermoMeccTrovato THEN
	            REGION Tempo OFF Marcia Motore
	                IF NOT "Motore".M[#K_MotoreInt].Dati.MotoreFermo THEN
	                    "Motore".M[#K_MotoreInt].Dati.ContTOffMotoreMarcia := 1000;
	                    "Motore".M[#K_MotoreInt].Dati.TOffMotoreMarcia := true;
	                ELSE
	                    IF "Motore".M[#K_MotoreInt].Dati.ContTOffMotoreMarcia > 0 THEN
	                        "Motore".M[#K_MotoreInt].Dati.ContTOffMotoreMarcia -= REAL_TO_INT("Zona".Comuni.TempoCicloCpu_r);
	                    ELSE
	                        "Motore".M[#K_MotoreInt].Dati.TOffMotoreMarcia := false;
	                    END_IF;
	                END_IF;
	            END_REGION ;
	            #REQSetup := "Motore".M[#K_MotoreInt].Dati.SetupFermoMeccTrovato AND NOT "Motore".M[#K_MotoreInt].Dati.TOffMotoreMarcia;
	            IF #REQSetup THEN
	                "Motore".M[#K_MotoreInt].Allarmi.SetupEncoderEseg := TRUE;
	            END_IF;
	            IF #REQSetup THEN
	                IF NOT "Motore".M[#K_MotoreInt].Dati.AppoImpEsecSetUP THEN
	                    "Motore".M[#K_MotoreInt].Dati.Encoder.ValoKSetupSuSens := "Motore".M[#K_MotoreInt].Out.ActPos - "Motore".M[#K_MotoreInt].Dati.PosImpulsoSetup;
	                    "Motore".M[#K_MotoreInt].Dati.AppoImpEsecSetUP := TRUE;
	                END_IF;
	            END_IF;
	            IF #REQSetup AND NOT #SetUpFermoMeccanico THEN
	                IF "Motore".M[#K_MotoreInt].Dati.ContSetUPEncoder > 300 THEN
	                    IF NOT #SetUpFermoMeccanico THEN
	                        "Motore".M[#K_MotoreInt].Dati.SetupFermoMeccTrovato := false;
	                    END_IF;
	                ELSE
	                    "Motore".M[#K_MotoreInt].Dati.ContSetUPEncoder += REAL_TO_INT("Zona".Comuni.TempoCicloCpu_r);
	                END_IF;
	            ELSE
	                "Motore".M[#K_MotoreInt].Dati.ContSetUPEncoder := 0;
	            END_IF;
	            IF NOT "Motore".M[#K_MotoreInt].Dati.SetupFermoMeccTrovato THEN
	                "Motore".M[#K_MotoreInt].Dati.AppoImpEsecSetUP := FALSE;
	                IF "Motore".M[#K_MotoreInt].Prm.Enc.SetupMode = 4 THEN
	                    "Motore".M[#K_MotoreInt].In.CmdPosRich := true;
	                    "Motore".M[#K_MotoreInt].In.CmdVelocitaRich := "Motore".M[#K_MotoreInt].Prm.VelSgancioFrenoPos;
	                    IF "Motore".M[#K_MotoreInt].Out.ActDirPos AND "Motore".M[#K_MotoreInt].Out.ActPos <= "Motore".M[#K_MotoreInt].Dati.MaxPosRicercaFermoMeccanico THEN
	                        "Motore".M[#K_MotoreInt].Dati.ContFermoMeccTrovato += REAL_TO_INT("Zona".Comuni.TempoCicloCpu_r);
	                    ELSE
	                        "Motore".M[#K_MotoreInt].Dati.MaxPosRicercaFermoMeccanico := "Motore".M[#K_MotoreInt].Out.ActPos;
	                        "Motore".M[#K_MotoreInt].Dati.ContFermoMeccTrovato := 0;
	                    END_IF;
	                ELSE
	                    "Motore".M[#K_MotoreInt].In.CmdNegRich := true;
	                    "Motore".M[#K_MotoreInt].In.CmdVelocitaRich := "Motore".M[#K_MotoreInt].Prm.VelSgancioFrenoNeg;
	                    IF "Motore".M[#K_MotoreInt].Out.ActDirNeg AND "Motore".M[#K_MotoreInt].Out.ActPos >= "Motore".M[#K_MotoreInt].Dati.MaxPosRicercaFermoMeccanico THEN
	                        "Motore".M[#K_MotoreInt].Dati.ContFermoMeccTrovato += REAL_TO_INT("Zona".Comuni.TempoCicloCpu_r);
	                    ELSE
	                        "Motore".M[#K_MotoreInt].Dati.MaxPosRicercaFermoMeccanico := "Motore".M[#K_MotoreInt].Out.ActPos;
	                        "Motore".M[#K_MotoreInt].Dati.ContFermoMeccTrovato := 0;
	                    END_IF;
	                END_IF;
	                "Motore".M[#K_MotoreInt].Dati.SetupFermoMeccTrovato := "Motore".M[#K_MotoreInt].Dati.ContFermoMeccTrovato > 500;
	                "Motore".M[#K_MotoreInt].Dati.PosImpulsoSetup := "Motore".M[#K_MotoreInt].Dati.MaxPosRicercaFermoMeccanico;
	                "Motore".M[#K_MotoreInt].Dati.ContCheckFollowError := 0;
	            ELSE
	                "Motore".M[#K_MotoreInt].In.CmdPosRich := "Motore".M[#K_MotoreInt].In.CmdNegRich := "Motore".M[#K_MotoreInt].In.Positioning := false;
	            END_IF;
	        END_IF;
	    END_REGION
	    REGION Gestione Encoder
	        (* Gestisco l'Allarme di Setup Eseguito per memorizzare su HMI l'esecuzione del Setuo*)
	        IF "Motore".M[#K_MotoreInt].Allarmi.SetupEncoderEseg THEN
	            "Motore".M[#K_MotoreInt].Dati.ContSegnSetup += REAL_TO_INT("Zona".Comuni.TempoCicloCpu_r);
	            IF "Motore".M[#K_MotoreInt].Dati.ContSegnSetup > 3000 THEN
	                "Motore".M[#K_MotoreInt].Allarmi.SetupEncoderEseg := false;
	                "Motore".M[#K_MotoreInt].Dati.ContSegnSetup := 0;
	            END_IF;
	        END_IF;
	        (* Una volta selezionato su HMI il Setup, se non avviene entro 3 secondi viene deselezionato *)
	        IF "Motore".M[#K_MotoreInt].HMI.Setup AND NOT #REQSetupPannello THEN
	            "Motore".M[#K_MotoreInt].Dati.ContTORichSetup += REAL_TO_INT("Zona".Comuni.TempoCicloCpu_r);
	            IF "Motore".M[#K_MotoreInt].Dati.ContTORichSetup > 3000 THEN
	                "Motore".M[#K_MotoreInt].HMI.Setup := false;
	            END_IF;
	        ELSE
	            "Motore".M[#K_MotoreInt].Dati.ContTORichSetup := 0;
	        END_IF;
	        IF NOT "Motore".M[#K_MotoreInt].Prm.Enc.EncoderLess THEN
	            (* Richiamo la gestione dell'Encoder *)
	            IF "Motore".M[#K_MotoreInt].Prm.Enc.Mounting <> 11 THEN
	                REGION CalcoloPosizioneSetup
	                    IF #REQSetup THEN
	                        CASE "Motore".M[#K_MotoreInt].Prm.Enc.SetupMode OF
	                            0: // Encoder HMI
	                                IF "Motore".M[#K_MotoreInt].Prm.Enc.SetupDoppio THEN
	                                    #TempEnc.AppoSetupRich := "Motore".M[#K_MotoreInt].HMI.ValoreSetupEncoder * 2;
	                                ELSE
	                                    #TempEnc.#AppoSetupRich := "Motore".M[#K_MotoreInt].HMI.ValoreSetupEncoder;
	                                END_IF;
	                                IF NOT "Motore".M[#K_MotoreInt].Prm.Enc.ModoCalcoloK THEN
	                                    "Motore".M[#K_MotoreInt].HMI.ValoreSetupRichiesto := "Motore".M[#K_MotoreInt].Prm.Enc.KSetup + #TempEnc.AppoSetupRich;
	                                ELSE
	                                    "Motore".M[#K_MotoreInt].HMI.ValoreSetupRichiesto := "Motore".M[#K_MotoreInt].Prm.Enc.KSetup - #TempEnc.AppoSetupRich;
	                                END_IF;
	                            1: // Encoder Esterno
	                                "Motore".M[#K_MotoreInt].HMI.ValoreSetupRichiesto := "Motore".M[#K_MotoreInt].In.ValoSetupEnc;
	                            2, 10: // Ricerca Sensore
	                                "Motore".M[#K_MotoreInt].HMI.ValoreSetupRichiesto := "Motore".M[#K_MotoreInt].HMI.ValoreSetupSensore + "Motore".M[#K_MotoreInt].Dati.Encoder.ValoKSetupSuSens;
	                            4, 12: // Ricerca Coppia
	                                "Motore".M[#K_MotoreInt].HMI.ValoreSetupRichiesto := "Motore".M[#K_MotoreInt].HMI.ValoreSetupSensore + "Motore".M[#K_MotoreInt].Dati.Encoder.ValoKSetupSuSens;
	                        END_CASE;
	                    END_IF;
	                END_REGION
	                REGION Lettura Encoder Dal Campo
	                    CASE "Motore".M[#K_MotoreInt].HW.TipoEncoder OF
	                        1:
	                            "Motore".M[#K_MotoreInt].Dati.Encoder.#RetValRdEnc := DPRD_DAT(LADDR := "Motore".M[#K_MotoreInt].HW.HWIO_Encoder, RECORD => #TempEnc.RcvDaEncoderSick);
	                            #TempEnc.#PosizioneLettaEnc := DWORD_TO_DINT(IN := SHR(IN := #TempEnc.RcvDaEncoderSick.Position01, N := 2));
	                            #TempEnc.VelocitaLettaEnc := #TempEnc.RcvDaEncoderSick.Speed;
	                            "Motore".M[#K_MotoreInt].Out.VelEncoder := ABS(TRUNC(DINT_TO_REAL(#TempEnc.VelocitaLettaEnc) * "Motore".M[#K_MotoreInt].Prm.C.SpazioGiroEncoder / "Motore".M[#K_MotoreInt].Prm.Enc.ImpRev * 100.0));
	                            IF (#TempEnc.RcvDaEncoderSick.G1_ZSW.%X15 OR #TempEnc.RcvDaEncoderSick.G1_ZSW.%X12) AND NOT #REQSetup THEN
	                                #TempEnc.SendAEncoderSick.G1_STW := 16#0000;
	                                #TempEnc.SendAEncoderSick.G1_STW.%X15 := #TempEnc.RcvDaEncoderSick.G1_ZSW.%X15;
	                                #TempEnc.SendAEncoderSick.STW2_ENC := 16#400;
	                                "Motore".M[#K_MotoreInt].Dati.Encoder.#RetValScrEnc := DPWR_DAT(LADDR := "Motore".M[#K_MotoreInt].HW.HWIO_Encoder, RECORD := #TempEnc.SendAEncoderSick);
	                            END_IF;
	                        9: // Sick Telemetrica
	                            "Motore".M[#K_MotoreInt].Prm.Enc.Mounting := USint#1;
	                            "Motore".M[#K_MotoreInt].Dati.Encoder.#RetValRdEnc := DPRD_DAT(LADDR := "Motore".M[#K_MotoreInt].HW.HWIO_Encoder, RECORD => #TempTelem.RcvDaEncoder);
	                            "Motore".M[#K_MotoreInt].Dati.Encoder.#RetValRdEnc := DPRD_DAT(LADDR := "Motore".M[#K_MotoreInt].HW.HWIO_PrmEncoder, RECORD => #TempTelem.RcvDaEncoder.Status);
	                            // Valore arriva in decimi di mm (*100 = converto in millesimi di millimetro)
	                            #TempEnc.#PosizioneLettaEnc := DWORD_TO_DINT(#TempTelem.RcvDaEncoder.M05_IN_ActPos * 100);
	                        10:
	                            "Motore".M[#K_MotoreInt].Dati.Encoder.#RetValRdEnc := DPRD_DAT(LADDR := "Motore".M[#K_MotoreInt].HW.HWIO_Encoder, RECORD => #TempEnc.#RcvDaEncoder_Ottico);
	                            #TempEnc.#PosizioneLettaEnc := #TempEnc.#RcvDaEncoder_Ottico.Posizione;
	                        11:
	                            "Motore".M[#K_MotoreInt].Dati.Encoder.#RetValRdEnc := DPRD_DAT(LADDR := "Motore".M[#K_MotoreInt].HW.HWIO_Encoder, RECORD => #TempEnc.#RcvDaEncoder_Magnetico);
	                            #TempEnc.#PosizioneLettaEnc := #TempEnc.#RcvDaEncoder_Magnetico.Posizione;
	                    END_CASE;
	                    "Motore".M[#K_MotoreInt].In.NoComunEnc := "Motore".M[#K_MotoreInt].Dati.Encoder.#RetValRdEnc <> 0 OR #TempEnc.#PosizioneLettaEnc = 0;
	                END_REGION
	                IF NOT "Motore".M[#K_MotoreInt].Prm.Mech.EndLess THEN
	                    REGION Gestione Encoder
	                        REGION CalcoloPosizione
	                            IF NOT "Motore".M[#K_MotoreInt].In.NoComunEnc THEN
	                                IF NOT "Motore".M[#K_MotoreInt].Prm.Enc.Direction THEN
	                                    IF "Motore".M[#K_MotoreInt].HW.TipoEncoder = 9 THEN
	                                        // Se Telemetrica (=9) Cambio Calcolo
	                                        IF #TempEnc.PosizioneLettaEnc <> 0 THEN
	                                            "Motore".M[#K_MotoreInt].Prm.C.EncPos := DINT_TO_REAL(#TempEnc.#PosizioneLettaEnc);
	                                        ELSE
	                                            "Motore".M[#K_MotoreInt].Allarmi.EncMismatch := true;
	                                        END_IF;
	                                    ELSE
	                                        "Motore".M[#K_MotoreInt].Prm.C.EncPos := DINT_TO_REAL(#TempEnc.PosizioneLettaEnc - "Motore".M[#K_MotoreInt].Dati.Encoder.MezzoRicircoloEncoder) / "Motore".M[#K_MotoreInt].Prm.Enc.ImpRev * "Motore".M[#K_MotoreInt].Prm.C.SpazioGiroEncoder;
	                                    END_IF;
	                                ELSE
	                                    IF "Motore".M[#K_MotoreInt].HW.TipoEncoder = 9 THEN
	                                        // Se Telemetrica (=9) Cambio Calcolo
	                                        IF #TempEnc.PosizioneLettaEnc <> 0 THEN
	                                            "Motore".M[#K_MotoreInt].Prm.C.EncPos := DINT_TO_REAL("Motore".M[#K_MotoreInt].Prm.Enc.KSetup - #TempEnc.#PosizioneLettaEnc);
	                                        ELSE
	                                            "Motore".M[#K_MotoreInt].Allarmi.EncMismatch := true;
	                                        END_IF;
	                                    ELSE
	                                        "Motore".M[#K_MotoreInt].Prm.C.EncPos := DINT_TO_REAL(- #TempEnc.PosizioneLettaEnc + "Motore".M[#K_MotoreInt].Dati.Encoder.MezzoRicircoloEncoder) / "Motore".M[#K_MotoreInt].Prm.Enc.ImpRev * "Motore".M[#K_MotoreInt].Prm.C.SpazioGiroEncoder;
	                                    END_IF;
	                                END_IF;
	                            END_IF;
	                        END_REGION
	                        REGION Gestione Setup Encoder
	                            IF #REQSetup THEN
	                                IF NOT "Motore".M[#K_MotoreInt].Dati.Encoder.RichSetupEnc THEN
	                                    "Motore".M[#K_MotoreInt].Out.EncoderHomed := false;
	                                END_IF;
	                                IF NOT "Motore".M[#K_MotoreInt].Prm.Enc.Direction THEN
	                                    #TempEnc.#AppoSetupEncoder := DINT_TO_UDINT(TRUNC(DINT_TO_REAL("Motore".M[#K_MotoreInt].HMI.ValoreSetupRichiesto) / "Motore".M[#K_MotoreInt].Prm.C.SpazioGiroEncoder * "Motore".M[#K_MotoreInt].Prm.Enc.ImpRev) + "Motore".M[#K_MotoreInt].Dati.Encoder.MezzoRicircoloEncoder);
	                                ELSE
	                                    #TempEnc.#AppoSetupEncoder := DINT_TO_UDINT(TRUNC(DINT_TO_REAL(- "Motore".M[#K_MotoreInt].HMI.ValoreSetupRichiesto) / "Motore".M[#K_MotoreInt].Prm.C.SpazioGiroEncoder * "Motore".M[#K_MotoreInt].Prm.Enc.ImpRev) + "Motore".M[#K_MotoreInt].Dati.Encoder.MezzoRicircoloEncoder);
	                                END_IF;
	                                IF "Motore".M[#K_MotoreInt].HW.TipoEncoder = 9 THEN
	                                    IF NOT "Motore".M[#K_MotoreInt].Prm.Enc.ModoCalcoloK THEN
	                                        #TempEnc.#AppoSetupEncoder := DINT_TO_UDINT("Motore".M[#K_MotoreInt].HMI.ValoreSetupRichiesto);
	                                    ELSE
	                                        #TempEnc.#AppoSetupEncoder := DINT_TO_UDINT("Motore".M[#K_MotoreInt].HMI.ValoreSetupEncoder);
	                                    END_IF;
	                                END_IF;
	                                IF #TempEnc.PosizioneLettaEnc <> #TempEnc.#AppoSetupEncoder OR #TempEnc.RcvDaEncoderSick.G1_ZSW.%X12 THEN
	                                    CASE "Motore".M[#K_MotoreInt].HW.TipoEncoder OF
	                                        1:
	                                            #TempEnc.#arrRecord[0] := 1;
	                                            #TempEnc.#arrRecord[1] := 2; (*Request ID = Change parameter*)
	                                            #TempEnc.#arrRecord[2] := 0; (*DO-ID*)
	                                            #TempEnc.#arrRecord[3] := 1; (*No. of parameters*)
	                                            #TempEnc.#arrRecord[4] := 16#10; (*Attribute = Value*)
	                                            #TempEnc.#arrRecord[5] := 0; (*No. of elements*)
	                                            #TempEnc.#arrRecord[6] := 16#fd; (*PNU high byte*)
	                                            #TempEnc.#arrRecord[7] := 16#e8; (*PNU low byte*)
	                                            #TempEnc.#arrRecord[8] := 0; (*Subindex high byte*)
	                                            #TempEnc.#arrRecord[9] := 0; (*Subindex low byte*)
	                                            #TempEnc.#arrRecord[10] := 16#43;
	                                            #TempEnc.#arrRecord[11] := 1;
	                                            #TempEnc.#arrRecord[12] := #TempEnc.#AppoSetupEncoder.%B3;
	                                            #TempEnc.#arrRecord[13] := #TempEnc.#AppoSetupEncoder.%B2;
	                                            #TempEnc.#arrRecord[14] := #TempEnc.#AppoSetupEncoder.%B1;
	                                            #TempEnc.#arrRecord[15] := #TempEnc.#AppoSetupEncoder.%B0;

	                              "WRREC"(REQ := "Motore".M[#K_MotoreInt].Dati.Encoder.RichSetupEnc AND NOT "Motore".M[#K_MotoreInt].Dati.SetupPN.Output.BUSY AND NOT "Motore".M[#K_MotoreInt].Dati.SetupPN.Output.DONE AND NOT "Motore".M[#K_MotoreInt].Dati.Encoder.PrmEncSend,
	                                      ID := "Motore".M[#K_MotoreInt].HW.HWIO_PrmEncoder,
	                                      INDEX := 16#B02E,
	                                      LEN := 16,
	                                      DONE => "Motore".M[#K_MotoreInt].Dati.SetupPN.Output.DONE,
	                                      BUSY => "Motore".M[#K_MotoreInt].Dati.SetupPN.Output.BUSY,
	                                      ERROR => "Motore".M[#K_MotoreInt].Dati.SetupPN.Output.ERROR,
	                                      STATUS => "Motore".M[#K_MotoreInt].Dati.SetupPN.Output.STATUS,
	                                      RECORD := #TempEnc.#arrRecord);

	                              IF "Motore".M[#K_MotoreInt].Dati.Encoder.RichSetupEnc THEN
	                                  IF "Motore".M[#K_MotoreInt].Dati.SetupPN.Output.DONE THEN
	                                                    "Motore".M[#K_MotoreInt].Dati.Encoder.PrmEncSend := true;
	                                                END_IF;
	                                            ELSE
	                                                "Motore".M[#K_MotoreInt].Dati.Encoder.PrmEncSend := false;
	                                            END_IF;
	                                            IF "Motore".M[#K_MotoreInt].Dati.Encoder.PrmEncSend AND NOT #TempEnc.RcvDaEncoderSick.G1_ZSW.%X12 THEN
	                                                #TempEnc.SendAEncoderSick.G1_STW := 16#1000;
	                                            ELSE
	                                                #TempEnc.SendAEncoderSick.G1_STW := 0;
	                                            END_IF;
	                                            #TempEnc.SendAEncoderSick.STW2_ENC := 16#400;
	                                            "Motore".M[#K_MotoreInt].Dati.Encoder.#RetValScrEnc := DPWR_DAT(LADDR := "Motore".M[#K_MotoreInt].HW.HWIO_Encoder, RECORD := #TempEnc.SendAEncoderSick);
	                                        9: // Setup Telemetrica
	                                            // Divido Valore per 100 per scrivere Valore in Decimi di mm
	                                            #TempTelem.SendAEncode.M05_OUT_Preset := UDINT_TO_DWORD(IN := #TempEnc.#AppoSetupEncoder / 100);
	                                            // Alzo bit richiesta Setup
	                                            #TempTelem.SendAEncode.M05_OUT_Preset.%X31 := TRUE;
	                                            "Motore".M[#K_MotoreInt].Dati.Encoder.#RetValScrEnc := DPWR_DAT(LADDR := "Motore".M[#K_MotoreInt].HW.HWIO_Encoder, RECORD := #TempTelem.SendAEncode);
	                                            "Motore".M[#K_MotoreInt].Dati.Encoder.#RichSetupEnc := true;
	                                        10:
	                                            #TempEnc.#AppoScrEncoder := (#TempEnc.#AppoSetupEncoder) OR dw#16#C0000000;

	                              "WRREC"(REQ := "Motore".M[#K_MotoreInt].Dati.Encoder.RichSetupEnc AND NOT "Motore".M[#K_MotoreInt].Dati.SetupPN.Output.BUSY AND NOT "Motore".M[#K_MotoreInt].Dati.SetupPN.Output.DONE,
	                                      ID := "Motore".M[#K_MotoreInt].HW.HWIO_PrmEncoder,
	                                      INDEX := 2,
	                                      LEN := 4,
	                                      DONE => "Motore".M[#K_MotoreInt].Dati.SetupPN.Output.DONE,
	                                      BUSY => "Motore".M[#K_MotoreInt].Dati.SetupPN.Output.BUSY,
	                                      ERROR => "Motore".M[#K_MotoreInt].Dati.SetupPN.Output.ERROR,
	                                      STATUS => "Motore".M[#K_MotoreInt].Dati.SetupPN.Output.STATUS,
	                                      RECORD := #TempEnc.AppoScrEncoder);

	                                        11:
	                                            #TempEnc.#AppoScrEncoder := #TempEnc.#AppoSetupEncoder;
	                                            "WRREC"(REQ := "Motore".M[#K_MotoreInt].Dati.Encoder.RichSetupEnc AND NOT "Motore".M[#K_MotoreInt].Dati.SetupPN.Output.BUSY AND NOT "Motore".M[#K_MotoreInt].Dati.SetupPN.Output.DONE,
	                                                    ID := "Motore".M[#K_MotoreInt].HW.HWIO_PrmEncoder,
	                                                    INDEX := 2,
	                                                    LEN := 4,
	                                                    DONE => "Motore".M[#K_MotoreInt].Dati.SetupPN.Output.DONE,
	                                                    BUSY => "Motore".M[#K_MotoreInt].Dati.SetupPN.Output.BUSY,
	                                                    ERROR => "Motore".M[#K_MotoreInt].Dati.SetupPN.Output.ERROR,
	                                                    STATUS => "Motore".M[#K_MotoreInt].Dati.SetupPN.Output.STATUS,
	                                                    RECORD := #TempEnc.AppoScrEncoder);

	                                    END_CASE;
	                                    "Motore".M[#K_MotoreInt].Dati.Encoder.#RichSetupEnc := true;
	                                ELSE
	                                    "Motore".M[#K_MotoreInt].Out.EncoderHomed := true;
	                                END_IF;
	                            ELSE
	                                IF "Motore".M[#K_MotoreInt].Dati.Encoder.RichSetupEnc THEN
	                                    CASE "Motore".M[#K_MotoreInt].HW.TipoEncoder OF
	                                        9:
	                                            #TempTelem.SendAEncode.M05_OUT_Preset := 0;
	                                            "Motore".M[#K_MotoreInt].Dati.Encoder.#RetValScrEnc := DPWR_DAT(LADDR := "Motore".M[#K_MotoreInt].HW.HWIO_Encoder, RECORD := #TempTelem.SendAEncode);
	                                    END_CASE;
	                                    "Motore".M[#K_MotoreInt].Dati.Encoder.RichSetupEnc := false;
	                                END_IF;
	                            END_IF;
	                        END_REGION
	                    END_REGION
	                ELSE
	                    REGION Gestione Encoder EndLess
	                        REGION Gestione Setup Encoder
	                            IF #REQSetup THEN
	                                "Motore".M[#K_MotoreInt].Out.EncoderHomed := true;
	                                "Motore".M[#K_MotoreInt].Prm.C.EncPos := DINT_TO_REAL("Motore".M[#K_MotoreInt].HMI.ValoreSetupRichiesto);
	                                "Motore".M[#K_MotoreInt].In.Setup := false;
	                            END_IF;
	                        END_REGION
	                        REGION REGION CalcoloPosizione
	                            IF NOT "Motore".M[#K_MotoreInt].In.NoComunEnc THEN
	                                #TempEnc.SpazioUltimoCiclo := #TempEnc.PosizioneLettaEnc - "Motore".M[#K_MotoreInt].Dati.Encoder.o_OldPosEncoder;
	                                IF #TempEnc.SpazioUltimoCiclo <> 0 THEN
	                                    IF ABS(#TempEnc.SpazioUltimoCiclo) > "Motore".M[#K_MotoreInt].Dati.Encoder.#MezzoRicircoloEncoder THEN
	                                        IF #TempEnc.PosizioneLettaEnc < "Motore".M[#K_MotoreInt].Dati.Encoder.o_OldPosEncoder THEN
	                                            #TempEnc.SpazioUltimoCiclo := "Motore".M[#K_MotoreInt].Dati.Encoder.#RicircoloEncoder - "Motore".M[#K_MotoreInt].Dati.Encoder.o_OldPosEncoder + #TempEnc.PosizioneLettaEnc;
	                                        ELSE
	                                            #TempEnc.SpazioUltimoCiclo := #TempEnc.PosizioneLettaEnc - "Motore".M[#K_MotoreInt].Dati.Encoder.#RicircoloEncoder - "Motore".M[#K_MotoreInt].Dati.Encoder.o_OldPosEncoder;
	                                        END_IF;
	                                    END_IF;
	                                    "Motore".M[#K_MotoreInt].Dati.Encoder.o_OldPosEncoder := #TempEnc.PosizioneLettaEnc;
	                                    IF NOT "Motore".M[#K_MotoreInt].Prm.Enc.Direction THEN
	                                        "Motore".M[#K_MotoreInt].Prm.C.EncPos += DINT_TO_REAL(#TempEnc.SpazioUltimoCiclo) * "Motore".M[#K_MotoreInt].Prm.C.SpazioGiroEncoder / "Motore".M[#K_MotoreInt].Prm.Enc.ImpRev;
	                                    ELSE
	                                        "Motore".M[#K_MotoreInt].Prm.C.EncPos -= DINT_TO_REAL(#TempEnc.SpazioUltimoCiclo) * "Motore".M[#K_MotoreInt].Prm.C.SpazioGiroEncoder / "Motore".M[#K_MotoreInt].Prm.Enc.ImpRev;
	                                    END_IF;
	                                    IF "Motore".M[#K_MotoreInt].Prm.C.EncPos > DINT_TO_REAL("Motore".M[#K_MotoreInt].Prm.Enc.ModuloPosEnc) THEN
	                                        "Motore".M[#K_MotoreInt].Prm.C.EncPos -= DINT_TO_REAL("Motore".M[#K_MotoreInt].Prm.Enc.ModuloPosEnc - "Motore".M[#K_MotoreInt].Prm.Enc.ModuloNegEnc);
	                                    ELSIF "Motore".M[#K_MotoreInt].Prm.C.EncPos < DINT_TO_REAL("Motore".M[#K_MotoreInt].Prm.Enc.ModuloNegEnc) THEN
	                                        "Motore".M[#K_MotoreInt].Prm.C.EncPos += DINT_TO_REAL("Motore".M[#K_MotoreInt].Prm.Enc.ModuloPosEnc - "Motore".M[#K_MotoreInt].Prm.Enc.ModuloNegEnc);
	                                    END_IF;
	                                END_IF;
	                            END_IF;
	                        END_REGION
	                    END_REGION
	                END_IF;
	            END_IF;
	            (* Assegnazione dati Posizione Encoder *)
	            "Motore".M[#K_MotoreInt].Out.ActPos := TRUNC("Motore".M[#K_MotoreInt].Prm.C.EncPos);
	            IF #REQSetup THEN
	                "Motore".M[#K_MotoreInt].Dati.PosizioneAlloStop := "Motore".M[#K_MotoreInt].Dati.PosizioneCheckDirezione := "Motore".M[#K_MotoreInt].Dati.TrgPosDint := "Motore".M[#K_MotoreInt].Dati.OldTrgPosDint := "Motore".M[#K_MotoreInt].Dati.OldEncoder := "Motore".M[#K_MotoreInt].Out.ActPos;
	                "Motore".M[#K_MotoreInt].Prm.C.TrgPos := "Motore".M[#K_MotoreInt].Prm.C.EncPos;
	            END_IF;
	        ELSIF #REQSetup THEN
	            (* Gestione Posizione Encoder Simulata *)
	            "Motore".M[#K_MotoreInt].Dati.PosizioneAlloStop := "Motore".M[#K_MotoreInt].Dati.PosizioneCheckDirezione := "Motore".M[#K_MotoreInt].Dati.TrgPosDint := "Motore".M[#K_MotoreInt].Dati.OldTrgPosDint := "Motore".M[#K_MotoreInt].Dati.OldEncoder := "Motore".M[#K_MotoreInt].Out.ActPos := "Motore".M[#K_MotoreInt].HMI.ValoreSetupEncoder;
	            "Motore".M[#K_MotoreInt].Prm.C.TrgPos := "Motore".M[#K_MotoreInt].Prm.C.EncPos := DINT_TO_REAL("Motore".M[#K_MotoreInt].HMI.ValoreSetupEncoder);
	            "Motore".M[#K_MotoreInt].In.Setup := false;
	        END_IF;
	    END_REGION
	    REGION Spazio Ciclo PLC
	        IF "Motore".M[#K_MotoreInt].Out.ActPos <> "Motore".M[#K_MotoreInt].Dati.OldEncoder THEN
	            "Motore".M[#K_MotoreInt].Out.SpazioCicloEnc := "Motore".M[#K_MotoreInt].Out.ActPos - "Motore".M[#K_MotoreInt].Dati.OldEncoder;
	            IF "Motore".M[#K_MotoreInt].Prm.Mech.EndLess THEN
	                IF ABS("Motore".M[#K_MotoreInt].Out.SpazioCicloEnc) > #MezzoRicircoloTotale THEN
	                    IF "Motore".M[#K_MotoreInt].Dati.OldEncoder > "Motore".M[#K_MotoreInt].Out.ActPos THEN
	                        "Motore".M[#K_MotoreInt].Out.SpazioCicloEnc := "Motore".M[#K_MotoreInt].Prm.Enc.ModuloPosEnc - "Motore".M[#K_MotoreInt].Dati.OldEncoder - "Motore".M[#K_MotoreInt].Prm.Enc.ModuloNegEnc + "Motore".M[#K_MotoreInt].Out.ActPos;
	                    ELSE
	                        "Motore".M[#K_MotoreInt].Out.SpazioCicloEnc := "Motore".M[#K_MotoreInt].Out.ActPos - "Motore".M[#K_MotoreInt].Prm.Enc.ModuloPosEnc + "Motore".M[#K_MotoreInt].Prm.Enc.ModuloNegEnc - "Motore".M[#K_MotoreInt].Dati.OldEncoder;
	                    END_IF;
	                END_IF;
	            END_IF;
	            "Motore".M[#K_MotoreInt].Dati.OldEncoder := "Motore".M[#K_MotoreInt].Out.ActPos;
	        ELSE
	            "Motore".M[#K_MotoreInt].Out.SpazioCicloEnc := 0;
	        END_IF;
	    END_REGION
	END_REGION ;
	REGION Limits
	    "Motore".M[#K_MotoreInt].Allarmi.Parametri := false;
	    REGION Abilita Cambio Direzione
	        IF "Motore".M[#K_MotoreInt].Prm.TCambioDir = 0 OR "Motore".M[#K_MotoreInt].Prm.CambioDirNoFreno THEN
	            #AbilDirPos := #AbilDirNeg := true;
	            "Motore".M[#K_MotoreInt].Dati.ContCambioDirPos := "Motore".M[#K_MotoreInt].Dati.ContCambioDirNeg := -1;
	        ELSE
	            IF "Motore".M[#K_MotoreInt].Out.ActDirNeg THEN
	                "Motore".M[#K_MotoreInt].Dati.ContCambioDirPos := "Motore".M[#K_MotoreInt].Prm.TCambioDir;
	            ELSIF "Motore".M[#K_MotoreInt].Out.ActDirPos THEN
	                "Motore".M[#K_MotoreInt].Dati.ContCambioDirNeg := "Motore".M[#K_MotoreInt].Prm.TCambioDir;
	            END_IF;
	            IF "Motore".M[#K_MotoreInt].Dati.ContCambioDirPos < 0 THEN
	                #AbilDirPos := true;
	            ELSE
	                "Motore".M[#K_MotoreInt].Dati.ContCambioDirPos -= REAL_TO_INT("Zona".Comuni.TempoCicloCpu_r);
	                #AbilDirPos := false;
	            END_IF;
	            IF "Motore".M[#K_MotoreInt].Dati.ContCambioDirNeg < 0 THEN
	                #AbilDirNeg := true;
	            ELSE
	                "Motore".M[#K_MotoreInt].Dati.ContCambioDirNeg -= REAL_TO_INT("Zona".Comuni.TempoCicloCpu_r);
	                #AbilDirNeg := false;
	            END_IF;
	        END_IF;
	    END_REGION
	    IF NOT "Motore".M[#K_MotoreInt].Prm.EscludiFunzPos THEN
	        REGION Abilita movimento motore / Posizionamento
	            "Motore".M[#K_MotoreInt].Out.Pronto := FALSE;
	            IF "Zona".Z[#K_Zona].Out.CentralinaOk THEN
	                IF NOT "Motore".M[#K_MotoreInt].In.SezAperto AND NOT "Motore".M[#K_MotoreInt].In.DriverFault AND NOT "Motore".M[#K_MotoreInt].In.NoComunInv THEN
	                    IF NOT "Motore".M[#K_MotoreInt].In.TerVentolaOff AND NOT "Motore".M[#K_MotoreInt].In.CinghiaRotta AND NOT "Motore".M[#K_MotoreInt].In.SpinaSicNoInPos AND ("Motore".M[#K_MotoreInt].In.AnticadutaON OR NOT "Motore".M[#K_MotoreInt].Prm.AnticadutaPresente) THEN
	                        "Motore".M[#K_MotoreInt].Out.Pronto := NOT "Motore".M[#K_MotoreInt].Dati.MotorStop;
	                    ELSIF "Zona".Z[#K_ZonaInt].Out.Man AND "Zona".Z[#K_ZonaInt].Gen.Reset AND ("Motore".M[#K_MotoreInt].In.CmdPosRich OR "Motore".M[#K_MotoreInt].In.CmdNegRich) THEN
	                        "Motore".M[#K_MotoreInt].Out.Pronto := TRUE;
	                    END_IF;
	                END_IF;
	            END_IF;
	            IF "Motore".M[#K_MotoreInt].In.Positioning THEN
	                #FunzPositioning := NOT "Motore".M[#K_MotoreInt].In.CmdPosRich AND NOT "Motore".M[#K_MotoreInt].In.CmdNegRich AND NOT #REQSetupPannello AND "Motore".M[#K_MotoreInt].Out.Pronto AND (NOT "Motore".M[#K_MotoreInt].In.NoComunEnc OR "Motore".M[#K_MotoreInt].Prm.Enc.EncoderLess);
	            ELSE
	                #FunzPositioning := FALSE;
	            END_IF;
	        END_REGION
	        REGION Controllo Limiti
	            IF "Motore".M[#K_MotoreInt].Prm.Mech.EndLess THEN
	(* In caso di Funzionamento EndLess, i limiti di posizione non possono superare gli estremi del ricircolo *)
	                "Motore".M[#K_MotoreInt].Prm.LimitePos := MIN(IN1 := "Motore".M[#K_MotoreInt].Prm.LimitePos, IN2 := "Motore".M[#K_MotoreInt].Prm.Enc.ModuloPosEnc);
	                "Motore".M[#K_MotoreInt].Prm.LimiteNeg := MAX(IN1 := "Motore".M[#K_MotoreInt].Prm.LimiteNeg, IN2 := "Motore".M[#K_MotoreInt].Prm.Enc.ModuloNegEnc);
	            END_IF;
	            IF "Motore".M[#K_MotoreInt].Prm.LimitePos <= "Motore".M[#K_MotoreInt].Prm.LimiteNeg THEN
	                "Motore".M[#K_MotoreInt].Prm.LimitePos := "Motore".M[#K_MotoreInt].Prm.LimiteNeg + 1;
	            END_IF;
	            IF "Motore".M[#K_MotoreInt].In.AttivaLimVarNeg THEN
	                "Motore".M[#K_MotoreInt].In.LimiteVarNeg := MIN(IN1 := "Motore".M[#K_MotoreInt].Prm.LimitePos, IN2 := "Motore".M[#K_MotoreInt].In.LimiteVarNeg);
	            END_IF;
	            IF "Motore".M[#K_MotoreInt].In.AttivaLimVarPos THEN
	                "Motore".M[#K_MotoreInt].In.LimiteVarPos := MAX(IN1 := "Motore".M[#K_MotoreInt].Prm.LimiteNeg, IN2 := "Motore".M[#K_MotoreInt].In.LimiteVarPos);
	            END_IF;
	            IF "Motore".M[#K_MotoreInt].In.AttivaLimVarNeg AND "Motore".M[#K_MotoreInt].In.AttivaLimVarPos THEN
	                IF "Motore".M[#K_MotoreInt].In.LimiteVarPos <= "Motore".M[#K_MotoreInt].In.LimiteVarNeg THEN
	                    "Motore".M[#K_MotoreInt].In.LimiteVarPos := "Motore".M[#K_MotoreInt].In.LimiteVarNeg + 1;
	                END_IF;
	            END_IF;
	        END_REGION
	        REGION Posizione Destinazione Assoluta/Relativa
	            "Motore".M[#K_MotoreInt].Allarmi.TrgPosMaxPos := "Motore".M[#K_MotoreInt].Allarmi.TrgPosMinNeg := "Motore".M[#K_MotoreInt].Allarmi.TrgPosMaxPosVar := "Motore".M[#K_MotoreInt].Allarmi.TrgPosMinNegVar := false;
	            IF "Motore".M[#K_MotoreInt].In.PosRelativo THEN
	                IF NOT "Motore".M[#K_MotoreInt].Dati.AppoImpMovRelativo THEN
	                    "Motore".M[#K_MotoreInt].Out.DistTRG := "Motore".M[#K_MotoreInt].Dati.MovRelRichiesto := "Motore".M[#K_MotoreInt].In.TrgPosRel;
	                END_IF;
	                IF NOT "Motore".M[#K_MotoreInt].Prm.Mech.EndLess THEN
	                    IF "Motore".M[#K_MotoreInt].Out.ActPos - "Motore".M[#K_MotoreInt].Out.DistTRG < "Motore".M[#K_MotoreInt].Prm.LimiteNeg THEN
	                        "Motore".M[#K_MotoreInt].Out.DistTRG := "Motore".M[#K_MotoreInt].Dati.MovRelRichiesto := "Motore".M[#K_MotoreInt].Out.ActPos - "Motore".M[#K_MotoreInt].Prm.LimiteNeg;
	                        IF #FunzPositioning THEN
	                            "Motore".M[#K_MotoreInt].Allarmi.Parametri := "Motore".M[#K_MotoreInt].Allarmi.TrgPosMinNeg := TRUE;
	                        END_IF;
	                    END_IF;
	                    IF "Motore".M[#K_MotoreInt].In.AttivaLimVarNeg THEN
	                        IF "Motore".M[#K_MotoreInt].Out.ActPos - "Motore".M[#K_MotoreInt].Out.DistTRG < "Motore".M[#K_MotoreInt].In.LimiteVarNeg THEN
	                            "Motore".M[#K_MotoreInt].Out.DistTRG := "Motore".M[#K_MotoreInt].Dati.MovRelRichiesto := "Motore".M[#K_MotoreInt].Out.ActPos - "Motore".M[#K_MotoreInt].In.LimiteVarNeg;
	                            IF #FunzPositioning THEN
	                                "Motore".M[#K_MotoreInt].Allarmi.Parametri := "Motore".M[#K_MotoreInt].Allarmi.TrgPosMinNegVar := TRUE;
	                            END_IF;
	                        END_IF;
	                    END_IF;
	                    IF "Motore".M[#K_MotoreInt].Out.ActPos + "Motore".M[#K_MotoreInt].Out.DistTRG > "Motore".M[#K_MotoreInt].Prm.LimitePos THEN
	                        "Motore".M[#K_MotoreInt].Out.DistTRG := "Motore".M[#K_MotoreInt].Dati.MovRelRichiesto := "Motore".M[#K_MotoreInt].Prm.LimitePos - "Motore".M[#K_MotoreInt].Out.ActPos;
	                        IF #FunzPositioning THEN
	                            "Motore".M[#K_MotoreInt].Allarmi.Parametri := "Motore".M[#K_MotoreInt].Allarmi.TrgPosMaxPos := TRUE;
	                        END_IF;
	                    END_IF;
	                    IF "Motore".M[#K_MotoreInt].In.AttivaLimVarPos THEN
	                        IF "Motore".M[#K_MotoreInt].Out.ActPos + "Motore".M[#K_MotoreInt].Out.DistTRG > "Motore".M[#K_MotoreInt].In.LimiteVarPos THEN
	                            "Motore".M[#K_MotoreInt].Out.DistTRG := "Motore".M[#K_MotoreInt].Dati.MovRelRichiesto := "Motore".M[#K_MotoreInt].In.LimiteVarPos - "Motore".M[#K_MotoreInt].Out.ActPos;
	                            IF #FunzPositioning THEN
	                                "Motore".M[#K_MotoreInt].Allarmi.Parametri := "Motore".M[#K_MotoreInt].Allarmi.TrgPosMaxPosVar := TRUE;
	                            END_IF;
	                        END_IF;
	                    END_IF;
	                    "Motore".M[#K_MotoreInt].Dati.MovRelRichiesto := ABS("Motore".M[#K_MotoreInt].Dati.MovRelRichiesto);
	                END_IF;
	            ELSE
	                "Motore".M[#K_MotoreInt].Out.TrgPosFiltrata := "Motore".M[#K_MotoreInt].In.TrgPos;
	                IF "Motore".M[#K_MotoreInt].Out.TrgPosFiltrata < "Motore".M[#K_MotoreInt].Prm.LimiteNeg THEN
	                    "Motore".M[#K_MotoreInt].Out.TrgPosFiltrata := "Motore".M[#K_MotoreInt].Prm.LimiteNeg;
	                    IF #FunzPositioning THEN
	                        "Motore".M[#K_MotoreInt].Allarmi.Parametri := "Motore".M[#K_MotoreInt].Allarmi.TrgPosMinNeg := TRUE;
	                    END_IF;
	                END_IF;
	                IF "Motore".M[#K_MotoreInt].In.AttivaLimVarNeg THEN
	                    IF "Motore".M[#K_MotoreInt].Out.TrgPosFiltrata < "Motore".M[#K_MotoreInt].In.LimiteVarNeg THEN
	                        "Motore".M[#K_MotoreInt].Out.TrgPosFiltrata := "Motore".M[#K_MotoreInt].In.LimiteVarNeg;
	                        IF #FunzPositioning THEN
	                            "Motore".M[#K_MotoreInt].Allarmi.Parametri := "Motore".M[#K_MotoreInt].Allarmi.TrgPosMinNegVar := TRUE;
	                        END_IF;
	                    END_IF;
	                END_IF;
	                IF "Motore".M[#K_MotoreInt].Out.TrgPosFiltrata > "Motore".M[#K_MotoreInt].Prm.LimitePos THEN
	                    "Motore".M[#K_MotoreInt].Out.TrgPosFiltrata := "Motore".M[#K_MotoreInt].Prm.LimitePos;
	                    IF #FunzPositioning THEN
	                        "Motore".M[#K_MotoreInt].Allarmi.Parametri := "Motore".M[#K_MotoreInt].Allarmi.TrgPosMaxPos := TRUE;
	                    END_IF;
	                END_IF;
	                IF "Motore".M[#K_MotoreInt].In.AttivaLimVarPos THEN
	                    IF "Motore".M[#K_MotoreInt].Out.TrgPosFiltrata > "Motore".M[#K_MotoreInt].In.LimiteVarPos THEN
	                        "Motore".M[#K_MotoreInt].Out.TrgPosFiltrata := "Motore".M[#K_MotoreInt].In.LimiteVarPos;
	                        IF #FunzPositioning THEN
	                            "Motore".M[#K_MotoreInt].Allarmi.Parametri := "Motore".M[#K_MotoreInt].Allarmi.TrgPosMaxPosVar := TRUE;
	                        END_IF;
	                    END_IF;
	                END_IF;
	            END_IF;
	            "Motore".M[#K_MotoreInt].Dati.AppoImpMovRelativo := "Motore".M[#K_MotoreInt].In.PosRelativo;
	        END_REGION
	        REGION Calcolo La Distanza Dal Target
	            IF NOT "Motore".M[#K_MotoreInt].In.PosRelativo THEN
	                "Motore".M[#K_MotoreInt].Out.DistTRG := "Motore".M[#K_MotoreInt].Out.TrgPosFiltrata - "Motore".M[#K_MotoreInt].Out.ActPos;
	                IF "Motore".M[#K_MotoreInt].Prm.Mech.EndLess THEN
	                    IF (#RicircoloTotale - "Motore".M[#K_MotoreInt].Out.DistTRG) < "Motore".M[#K_MotoreInt].Prm.Precisione THEN
	                        "Motore".M[#K_MotoreInt].Out.DistTRG := #RicircoloTotale - "Motore".M[#K_MotoreInt].Out.DistTRG;
	                    END_IF;
	                    IF #RicircoloTotale + "Motore".M[#K_MotoreInt].Out.DistTRG < "Motore".M[#K_MotoreInt].Prm.Precisione THEN
	                        "Motore".M[#K_MotoreInt].Out.DistTRG := #RicircoloTotale + "Motore".M[#K_MotoreInt].Out.DistTRG;
	                    END_IF;
	                    IF "Motore".M[#K_MotoreInt].In.ForzaEndLessPos THEN
	                        IF "Motore".M[#K_MotoreInt].Out.DistTRG < - "Motore".M[#K_MotoreInt].Prm.Precisione THEN
	                            "Motore".M[#K_MotoreInt].Out.DistTRG := "Motore".M[#K_MotoreInt].Out.DistTRG + #RicircoloTotale;
	                        END_IF;
	                    ELSIF "Motore".M[#K_MotoreInt].In.ForzaEndLessNeg THEN
	                        IF "Motore".M[#K_MotoreInt].Out.DistTRG > "Motore".M[#K_MotoreInt].Prm.Precisione THEN
	                            "Motore".M[#K_MotoreInt].Out.DistTRG := "Motore".M[#K_MotoreInt].Out.DistTRG - #RicircoloTotale;
	                        END_IF;
	                    ELSIF "Motore".M[#K_MotoreInt].In.ForzaEndLessBreve THEN
	                        IF "Motore".M[#K_MotoreInt].Out.DistTRG > #MezzoRicircoloTotale THEN
	                            "Motore".M[#K_MotoreInt].Out.DistTRG := "Motore".M[#K_MotoreInt].Out.DistTRG - #RicircoloTotale;
	                        ELSIF "Motore".M[#K_MotoreInt].Out.DistTRG < - #MezzoRicircoloTotale THEN
	                            "Motore".M[#K_MotoreInt].Out.DistTRG := "Motore".M[#K_MotoreInt].Out.DistTRG + #RicircoloTotale;
	                        END_IF;
	                    END_IF;
	                END_IF;
	            ELSE
	                "Motore".M[#K_MotoreInt].Out.DistTRG -= "Motore".M[#K_MotoreInt].Out.SpazioCicloEnc;
	            END_IF;
	            #DistTRG_ASS := ABS("Motore".M[#K_MotoreInt].Out.DistTRG);
	        END_REGION
	        REGION Time-Out Motore in Posizione
	            #DistTrgMagPrec := "Motore".M[#K_MotoreInt].Out.DistTRG > "Motore".M[#K_MotoreInt].Prm.Precisione;
	            #DistTrgMinPrec := "Motore".M[#K_MotoreInt].Out.DistTRG < - "Motore".M[#K_MotoreInt].Prm.Precisione;
	            IF NOT #DistTrgMagPrec AND NOT #DistTrgMinPrec THEN
	                IF "Motore".M[#K_MotoreInt].Dati.ContMotoreInPrec < 2000 THEN
	                    "Motore".M[#K_MotoreInt].Dati.ContMotoreInPrec += REAL_TO_INT("Zona".Comuni.TempoCicloCpu_r);
	                ELSE
	                    #RitMotInPrecisione := true;
	                END_IF;
	            ELSE
	                #RitMotInPrecisione := FALSE;
	                "Motore".M[#K_MotoreInt].Dati.ContMotoreInPrec := 0;
	            END_IF;
	        END_REGION
	        REGION Direzione Richiesta da Posizionatore
	            IF "Motore".M[#K_MotoreInt].Out.DistTRG > "Motore".M[#K_MotoreInt].Prm.SpazioArrestoPos THEN
	                IF #DistTrgMagPrec THEN
	                    "Motore".M[#K_MotoreInt].Out.RichMovPos := TRUE;
	                ELSIF #RitMotInPrecisione THEN
	                    "Motore".M[#K_MotoreInt].Out.RichMovPos := FALSE;
	                END_IF;
	                "Motore".M[#K_MotoreInt].Out.RichMovNeg := FALSE;
	                "Motore".M[#K_MotoreInt].Out.PosOK := NOT "Motore".M[#K_MotoreInt].Out.RichMovPos;
	            ELSIF "Motore".M[#K_MotoreInt].Out.DistTRG < - "Motore".M[#K_MotoreInt].Prm.SpazioArrestoNeg THEN
	                IF #DistTrgMinPrec THEN
	                    "Motore".M[#K_MotoreInt].Out.RichMovNeg := TRUE;
	                ELSIF #RitMotInPrecisione THEN
	                    "Motore".M[#K_MotoreInt].Out.RichMovNeg := FALSE;
	                END_IF;
	                "Motore".M[#K_MotoreInt].Out.RichMovPos := FALSE;
	                "Motore".M[#K_MotoreInt].Out.PosOK := NOT "Motore".M[#K_MotoreInt].Out.RichMovNeg;
	            ELSE
	                "Motore".M[#K_MotoreInt].Out.RichMovPos := FALSE;
	                "Motore".M[#K_MotoreInt].Out.RichMovNeg := FALSE;
	                "Motore".M[#K_MotoreInt].Out.PosOK := TRUE;
	            END_IF;
	        END_REGION
	        REGION Adattamento Perc.In Lavoro
	            #CambioPercLavoro := "Motore".M[#K_MotoreInt].Dati.Memo_PercentualeRich <> "Motore".M[#K_MotoreInt].In.PercentualeRichiesta;
	            IF #CambioPercLavoro THEN
	                IF "Motore".M[#K_MotoreInt].In.PercentualeRichiesta < 20 OR "Motore".M[#K_MotoreInt].In.PercentualeRichiesta > 100 THEN
	                    "Motore".M[#K_MotoreInt].In.PercentualeRichiesta := 100;
	                END_IF;
	                "Motore".M[#K_MotoreInt].Dati.Memo_PercentualeRich := "Motore".M[#K_MotoreInt].In.PercentualeRichiesta;
	            END_IF;
	(* Controllo cambio VelocitÃ  Richiesta *)
	            #CambioReqVel := "Motore".M[#K_MotoreInt].Dati.Memo_Req_Vel <> "Motore".M[#K_MotoreInt].In.CmdVelocitaRich OR #CambioPercLavoro OR "Motore".M[#K_MotoreInt].Allarmi.TrgVelMinFreno OR "Motore".M[#K_MotoreInt].Allarmi.TrgVelMaxMax;
	            IF #CambioReqVel THEN
	                "Motore".M[#K_MotoreInt].Dati.Memo_Req_Vel := "Motore".M[#K_MotoreInt].In.CmdVelocitaRich;
	                "Motore".M[#K_MotoreInt].Dati.VeloRichPerc := "Motore".M[#K_MotoreInt].Dati.Memo_Req_Vel * "Motore".M[#K_MotoreInt].In.PercentualeRichiesta / DINT#100;
	            END_IF;
	(* Controllo Cambio Accelerazione richiesta *)
	            #CambioReqAcc := "Motore".M[#K_MotoreInt].Dati.Memo_Req_Acc <> "Motore".M[#K_MotoreInt].In.Acc OR #CambioPercLavoro OR "Motore".M[#K_MotoreInt].Allarmi.AccRichZero OR "Motore".M[#K_MotoreInt].Allarmi.AccRichMaxMaxDec;
	            IF #CambioReqAcc THEN
	                "Motore".M[#K_MotoreInt].Dati.Memo_Req_Acc := MAX(IN1 := "Motore".M[#K_MotoreInt].In.Acc, IN2 := 10);
	                "Motore".M[#K_MotoreInt].Dati.AccRichPerc := "Motore".M[#K_MotoreInt].Dati.Memo_Req_Acc * "Motore".M[#K_MotoreInt].In.PercentualeRichiesta / DINT#100;
	            END_IF;
	(* Controllo Cambio Decelerazione richiesta *)
	            #CambioReqDec := "Motore".M[#K_MotoreInt].Dati.Memo_Req_Dec <> "Motore".M[#K_MotoreInt].In.Dec OR #CambioPercLavoro OR "Motore".M[#K_MotoreInt].Allarmi.DecRichZero OR "Motore".M[#K_MotoreInt].Allarmi.DecRichMaxMaxDec;
	            IF #CambioReqDec THEN
	                "Motore".M[#K_MotoreInt].Dati.Memo_Req_Dec := MAX(IN1 := "Motore".M[#K_MotoreInt].In.Dec, IN2 := 10);
	                "Motore".M[#K_MotoreInt].Dati.DecRichPerc := "Motore".M[#K_MotoreInt].Dati.Memo_Req_Dec * "Motore".M[#K_MotoreInt].In.PercentualeRichiesta / DINT#100;
	            END_IF;
	        END_REGION
	        #VeloBassaConv := DINT_TO_REAL("Motore".M[#K_MotoreInt].Prm.VelBassa);
	        REGION Direzione Movimento Richiesta
	            IF ("Motore".M[#K_MotoreInt].Out.RichMovPos AND "Motore".M[#K_MotoreInt].In.ConsMovimentoPos AND #FunzPositioning OR "Motore".M[#K_MotoreInt].In.CmdPosRich) AND "Motore".M[#K_MotoreInt].Out.Pronto AND #AbilDirPos THEN
	                #ReqDirPos := TRUE;
	                #ReqDirNeg := FALSE;
	                #UnaDirezioneRichiesta := TRUE;
	            ELSIF ("Motore".M[#K_MotoreInt].Out.RichMovNeg AND "Motore".M[#K_MotoreInt].In.ConsMovimentoNeg AND #FunzPositioning OR "Motore".M[#K_MotoreInt].In.CmdNegRich) AND "Motore".M[#K_MotoreInt].Out.Pronto AND #AbilDirNeg THEN
	                #ReqDirPos := FALSE;
	                #ReqDirNeg := TRUE;
	                #UnaDirezioneRichiesta := TRUE;
	            ELSE
	                #ReqDirPos := FALSE;
	                #ReqDirNeg := FALSE;
	                #UnaDirezioneRichiesta := FALSE;
	            END_IF;
	        END_REGION
	        REGION Posizione PiÃ¹ e Meno Inerzia
	            "Motore".M[#K_MotoreInt].Out.ActPosPiuInerzia := "Motore".M[#K_MotoreInt].Out.ActPos + "Motore".M[#K_MotoreInt].Prm.Inerzia;
	            "Motore".M[#K_MotoreInt].Out.ActPosMenoInerzia := "Motore".M[#K_MotoreInt].Out.ActPos - "Motore".M[#K_MotoreInt].Prm.Inerzia;
	            "Motore".M[#K_MotoreInt].Out.MinTrg := "Motore".M[#K_MotoreInt].Out.DistTRG > "Motore".M[#K_MotoreInt].Prm.Inerzia;
	            "Motore".M[#K_MotoreInt].Out.MaxTrg := "Motore".M[#K_MotoreInt].Out.DistTRG < - "Motore".M[#K_MotoreInt].Prm.Inerzia;
	            "Motore".M[#K_MotoreInt].Out.ActInInerzia := NOT "Motore".M[#K_MotoreInt].Out.MinTrg AND NOT "Motore".M[#K_MotoreInt].Out.MaxTrg;
	            IF "Motore".M[#K_MotoreInt].Prm.Mech.EndLess THEN
	                IF "Motore".M[#K_MotoreInt].Out.ActPosMenoInerzia < "Motore".M[#K_MotoreInt].Prm.Enc.ModuloNegEnc THEN
	                    "Motore".M[#K_MotoreInt].Out.ActPosMenoInerzia += #RicircoloTotale;
	                END_IF;
	                IF "Motore".M[#K_MotoreInt].Out.ActPosPiuInerzia > "Motore".M[#K_MotoreInt].Prm.Enc.ModuloPosEnc THEN
	                    "Motore".M[#K_MotoreInt].Out.ActPosPiuInerzia -= #RicircoloTotale;
	                END_IF;
	            END_IF;
	            "Motore".M[#K_MotoreInt].Out.MaxLimPos := "Motore".M[#K_MotoreInt].Out.ActPosPiuInerzia >= "Motore".M[#K_MotoreInt].Prm.LimitePos;
	            "Motore".M[#K_MotoreInt].Out.MinLimNeg := "Motore".M[#K_MotoreInt].Out.ActPosMenoInerzia <= "Motore".M[#K_MotoreInt].Prm.LimiteNeg;
	        END_REGION
	    ELSE
	        REGION Abilita movimento motore
	            "Motore".M[#K_MotoreInt].Out.Pronto := FALSE;
	            IF "Zona".Z[#K_Zona].Out.CentralinaOk THEN
	                IF NOT "Motore".M[#K_MotoreInt].In.SezAperto AND NOT "Motore".M[#K_MotoreInt].In.DriverFault AND NOT "Motore".M[#K_MotoreInt].In.NoComunInv AND NOT "Motore".M[#K_MotoreInt].In.TerVentolaOff THEN
	                    "Motore".M[#K_MotoreInt].Out.Pronto := TRUE;
	                END_IF;
	            END_IF;
	            #FunzPositioning := FALSE;

